KUKA KRL program: MyProgram_215().src

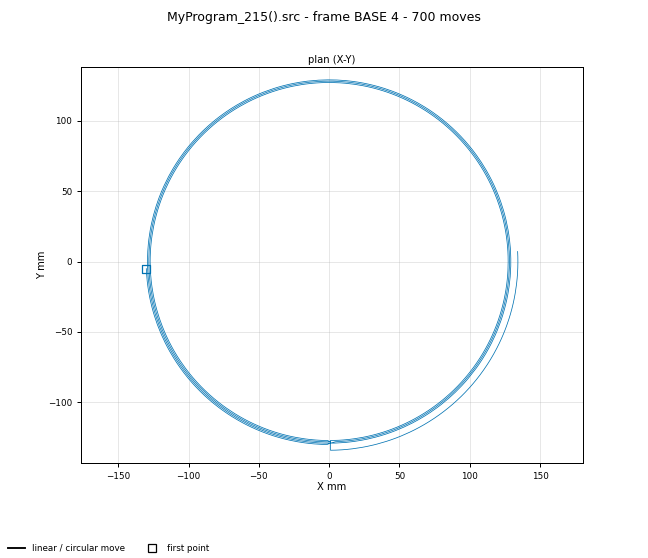
[picture p0: tool path of MyProgram_215().src in frame BASE 4, 700 of 700 moves have a stored position in this frame; points joined in program order, loops and branches not executed]
&ACCESS RVP
&REL 1
&PARAM TEMPLATE = C:\KRC\Roboter\Template\vorgabe
&PARAM EDITMASK = *
DEF MyProgram_215()
; ---- Setting reference (Base) ----
$BASE = BASE_DATA[4]

; --------------------------
; ---- Setting tool (TCP) ----
$TOOL = TOOL_DATA[3]
; --------------------------

$VEL.CP = VEL_APROX_PRINT
Startdeposition()
$VEL.CP = VEL_PRINT
LIN {X -130.0053,Y -5.0673,Z 151,A 179.9442,B 21.842,C -0.957,E1 21.7019,E2 267.4478} C_DIS
LIN {X -129.8507,Y -8.1164,Z 151,A -178.6124,B 21.842,C -0.9568,E1 21.7021,E2 265.9949} C_DIS
LIN {X -129.3313,Y -14.1597,Z 151,A -175.7971,B 21.8421,C -0.9542,E1 21.7029,E2 263.1669} C_DIS
LIN {X -128.8649,Y -17.9196,Z 151,A -174.1689,B 21.8424,C -0.9473,E1 21.7035,E2 261.5461} C_DIS
LIN {X -128.3149,Y -21.5014,Z 151,A -172.6656,B 21.8428,C -0.9385,E1 21.7041,E2 260.0561} C_DIS
LIN {X -127.7529,Y -24.622,Z 151,A -171.2515,B 21.8429,C -0.9349,E1 21.7049,E2 258.6421} C_DIS
LIN {X -127.1006,Y -27.7949,Z 151,A -169.6773,B 21.8429,C -0.9366,E1 21.7058,E2 257.0526} C_DIS
LIN {X -126.1184,Y -31.9552,Z 151,A -167.8984,B 21.8433,C -0.9266,E1 21.707,E2 255.2887} C_DIS
LIN {X -125.2346,Y -35.2609,Z 151,A -166.3979,B 21.8435,C -0.9217,E1 21.7081,E2 253.7911} C_DIS
LIN {X -124.2723,Y -38.5171,Z 151,A -164.8134,B 21.8435,C -0.9209,E1 21.7094,E2 252.1982} C_DIS
LIN {X -122.0887,Y -44.9645,Z 151,A -161.9059,B 21.844,C -0.9083,E1 21.712,E2 249.3057} C_DIS
LIN {X -120.3033,Y -49.5427,Z 151,A -159.7544,B 21.8443,C -0.9015,E1 21.7142,E2 247.1586} C_DIS
LIN {X -119.3188,Y -51.8654,Z 151,A -158.5882,B 21.8443,C -0.9006,E1 21.7155,E2 245.9873} C_DIS
LIN {X -117.9739,Y -54.8558,Z 151,A -157.1185,B 21.8444,C -0.8976,E1 21.7172,E2 244.5164} C_DIS
LIN {X -116.6239,Y -57.6698,Z 151,A -155.732,B 21.8446,C -0.8942,E1 21.7189,E2 243.1302} C_DIS
LIN {X -115.0398,Y -60.7689,Z 151,A -153.8793,B 21.8442,C -0.9033,E1 21.7214,E2 241.2414} C_DIS
LIN {X -113.4726,Y -63.6497,Z 151,A -152.4287,B 21.8443,C -0.8997,E1 21.7233,E2 239.7918} C_DIS
LIN {X -111.8624,Y -66.4401,Z 151,A -151.4946,B 21.8453,C -0.8757,E1 21.7246,E2 238.9168} C_DIS
LIN {X -110.3326,Y -68.9508,Z 151,A -149.9036,B 21.8449,C -0.8847,E1 21.727,E2 237.2922} C_DIS
LIN {X -108.359,Y -72.0127,Z 151,A -148.2536,B 21.845,C -0.8825,E1 21.7295,E2 235.6385} C_DIS
LIN {X -105.7262,Y -75.825,Z 151,A -146.2343,B 21.8452,C -0.8765,E1 21.7327,E2 233.6238} C_DIS
LIN {X -103.0748,Y -79.3925,Z 151,A -144.2157,B 21.8453,C -0.8743,E1 21.7361,E2 231.6} C_DIS
LIN {X -100.2325,Y -82.9511,Z 151,A -142.2432,B 21.8456,C -0.8682,E1 21.7396,E2 229.6333} C_DIS
LIN {X -97.3714,Y -86.2918,Z 151,A -140.1894,B 21.8456,C -0.8687,E1 21.7434,E2 227.5674} C_DIS
LIN {X -94.8101,Y -89.0985,Z 151,A -138.5955,B 21.8458,C -0.8616,E1 21.7464,E2 225.9844} C_DIS
LIN {X -91.7544,Y -92.2419,Z 151,A -136.1731,B 21.8452,C -0.8785,E1 21.7513,E2 223.5046} C_DIS
LIN {X -88.3402,Y -95.5175,Z 151,A -134.5958,B 21.8461,C -0.8526,E1 21.7544,E2 221.9896} C_DIS
LIN {X -85.1915,Y -98.3361,Z 151,A -132.7072,B 21.8462,C -0.8501,E1 21.7584,E2 220.0991} C_DIS
LIN {X -81.9083,Y -101.0868,Z 151,A -130.7823,B 21.8463,C -0.8482,E1 21.7625,E2 218.1708} C_DIS
LIN {X -78.3266,Y -103.8864,Z 151,A -128.5806,B 21.8461,C -0.8532,E1 21.7675,E2 215.9463} C_DIS
LIN {X -75.6688,Y -105.8379,Z 151,A -127.3113,B 21.8465,C -0.8429,E1 21.7703,E2 214.6997} C_DIS
LIN {X -72.1973,Y -108.2357,Z 151,A -125.4781,B 21.8466,C -0.8388,E1 21.7745,E2 212.8705} C_DIS
LIN {X -69.0452,Y -110.2738,Z 151,A -123.8621,B 21.8468,C -0.8347,E1 21.7783,E2 211.2596} C_DIS
LIN {X -65.5088,Y -112.4107,Z 151,A -121.9616,B 21.8468,C -0.8355,E1 21.7829,E2 209.3502} C_DIS
LIN {X -61.4607,Y -114.6736,Z 151,A -119.7151,B 21.8465,C -0.8416,E1 21.7885,E2 207.0798} C_DIS
LIN {X -58.5733,Y -116.1738,Z 151,A -118.6176,B 21.8471,C -0.8253,E1 21.7911,E2 206.023} C_DIS
LIN {X -55.1563,Y -117.835,Z 151,A -116.7367,B 21.8469,C -0.8323,E1 21.7959,E2 204.1176} C_DIS
LIN {X -51.0969,Y -119.6511,Z 151,A -114.7006,B 21.8469,C -0.8335,E1 21.8011,E2 202.0725} C_DIS
LIN {X -46.9474,Y -121.3381,Z 151,A -112.9585,B 21.8473,C -0.8215,E1 21.8056,E2 200.3584} C_DIS
LIN {X -42.9787,Y -122.8004,Z 151,A -111.0488,B 21.8473,C -0.8219,E1 21.8106,E2 198.4432} C_DIS
LIN {X -39.5704,Y -123.9401,Z 151,A -109.5332,B 21.8474,C -0.8177,E1 21.8146,E2 196.9357} C_DIS
LIN {X -36.3158,Y -124.9328,Z 151,A -108.0119,B 21.8474,C -0.8177,E1 21.8187,E2 195.4116} C_DIS
LIN {X -32.514,Y -125.9766,Z 151,A -105.7713,B 21.8466,C -0.8389,E1 21.8249,E2 193.1101} C_DIS
LIN {X -28.2456,Y -127.0028,Z 151,A -104.3076,B 21.8474,C -0.8171,E1 21.8288,E2 191.7029} C_DIS
LIN {X -22.4235,Y -128.1579,Z 151,A -101.5355,B 21.8472,C -0.823,E1 21.8364,E2 188.9112} C_DIS
LIN {X -18.2657,Y -128.8154,Z 151,A -99.8848,B 21.8476,C -0.8135,E1 21.8409,E2 187.2845} C_DIS
LIN {X -14.3497,Y -129.3109,Z 151,A -97.7475,B 21.8469,C -0.8311,E1 21.847,E2 185.0985} C_DIS
LIN {X -10.6851,Y -129.6647,Z 151,A -96.279,B 21.8472,C -0.8241,E1 21.851,E2 183.6479} C_DIS
LIN {X -5.5701,Y -129.9857,Z 151,A -94.1837,B 21.8474,C -0.8169,E1 21.8568,E2 181.5713} C_DIS
LIN {X -1.5263,Y -130.0967,Z 151,A -92.0677,B 21.8469,C -0.8323,E1 21.8628,E2 179.414} C_DIS
LIN {X -1.5263,Y -130.0967,Z 151,A -92.0677,B 21.8469,C -0.8323,E1 21.8628,E2 179.414} C_DIS
Enddeposition()
LIN {X 0.9297,Y -129.1307,Z 151,A -91.5034,B 20.7332,C -0.6398,E1 20.7439,E2 179.2548} C_DIS
Startdeposition()
$VEL.CP = VEL_PRINT
LIN {X -3.6627,Y -129.1076,Z 151,A -93.7153,B 20.7334,C -0.6318,E1 20.7376,E2 181.4893} C_DIS
LIN {X -8.0279,Y -128.9098,Z 151,A -95.6805,B 20.7334,C -0.6306,E1 20.7322,E2 183.4585} C_DIS
LIN {X -14.7037,Y -128.3212,Z 151,A -98.7805,B 20.7336,C -0.6256,E1 20.7235,E2 186.5747} C_DIS
LIN {X -20.0176,Y -127.599,Z 151,A -100.965,B 20.7333,C -0.6342,E1 20.7175,E2 188.7369} C_DIS
LIN {X -23.6572,Y -126.9757,Z 151,A -102.7964,B 20.7335,C -0.6269,E1 20.7124,E2 190.5914} C_DIS
LIN {X -28.0811,Y -126.0716,Z 151,A -105.0426,B 20.7338,C -0.6179,E1 20.7062,E2 192.8664} C_DIS
LIN {X -31.2653,Y -125.3191,Z 151,A -106.2307,B 20.7335,C -0.6294,E1 20.7031,E2 194.0238} C_DIS
LIN {X -34.6603,Y -124.4218,Z 151,A -107.7187,B 20.7333,C -0.6333,E1 20.6991,E2 195.5037} C_DIS
LIN {X -37.6238,Y -123.558,Z 151,A -109.1075,B 20.7333,C -0.6335,E1 20.6953,E2 196.8949} C_DIS
LIN {X -40.9396,Y -122.4992,Z 151,A -110.671,B 20.7333,C -0.6339,E1 20.6912,E2 198.4607} C_DIS
LIN {X -44.9395,Y -121.0895,Z 151,A -112.5539,B 20.7333,C -0.6355,E1 20.6862,E2 200.3437} C_DIS
LIN {X -49.6607,Y -119.2304,Z 151,A -114.8055,B 20.7333,C -0.6377,E1 20.6804,E2 202.595} C_DIS
LIN {X -53.9707,Y -117.3426,Z 151,A -116.9258,B 20.7332,C -0.6387,E1 20.675,E2 204.7188} C_DIS
LIN {X -56.9619,Y -115.9199,Z 151,A -118.3817,B 20.7332,C -0.641,E1 20.6713,E2 206.1728} C_DIS
LIN {X -62.2333,Y -113.18,Z 151,A -121.1366,B 20.7332,C -0.6397,E1 20.6645,E2 208.941} C_DIS
LIN {X -66.0389,Y -111.0019,Z 151,A -122.937,B 20.7329,C -0.6482,E1 20.6602,E2 210.7237} C_DIS
LIN {X -69.6038,Y -108.802,Z 151,A -124.8823,B 20.7329,C -0.6476,E1 20.6556,E2 212.6785} C_DIS
LIN {X -73.1285,Y -106.4649,Z 151,A -126.7619,B 20.7329,C -0.6505,E1 20.6512,E2 214.5576} C_DIS
LIN {X -77.9911,Y -102.9563,Z 151,A -129.4785,B 20.7328,C -0.6528,E1 20.6451,E2 217.2795} C_DIS
LIN {X -81.4308,Y -100.2583,Z 151,A -131.4493,B 20.7328,C -0.6551,E1 20.6408,E2 219.2528} C_DIS
LIN {X -84.7969,Y -97.4272,Z 151,A -133.3793,B 20.7326,C -0.6596,E1 20.6367,E2 221.1791} C_DIS
LIN {X -87.2832,Y -95.2062,Z 151,A -135.0805,B 20.7327,C -0.6539,E1 20.6331,E2 222.9049} C_DIS
LIN {X -89.6382,Y -92.9921,Z 151,A -136.651,B 20.7328,C -0.6515,E1 20.63,E2 224.4901} C_DIS
LIN {X -92.4164,Y -90.2322,Z 151,A -137.976,B 20.7322,C -0.6712,E1 20.6275,E2 225.7662} C_DIS
LIN {X -94.6886,Y -87.8446,Z 151,A -139.5529,B 20.7322,C -0.6699,E1 20.6244,E2 227.3553} C_DIS
LIN {X -97.6329,Y -84.5606,Z 151,A -141.5197,B 20.7322,C -0.6739,E1 20.6208,E2 229.3216} C_DIS
LIN {X -100.4671,Y -81.1722,Z 151,A -143.4289,B 20.7319,C -0.6804,E1 20.6174,E2 231.2232} C_DIS
LIN {X -103.0369,Y -77.8843,Z 151,A -145.3108,B 20.7319,C -0.6837,E1 20.6142,E2 233.107} C_DIS
LIN {X -105.6551,Y -74.2939,Z 151,A -147.2947,B 20.7317,C -0.688,E1 20.611,E2 235.0904} C_DIS
LIN {X -108.1691,Y -70.5839,Z 151,A -149.3281,B 20.7316,C -0.6913,E1 20.6078,E2 237.127} C_DIS
LIN {X -110.4376,Y -66.9785,Z 151,A -151.1709,B 20.7314,C -0.698,E1 20.6051,E2 238.9624} C_DIS
LIN {X -111.9833,Y -64.3618,Z 151,A -153.0329,B 20.7319,C -0.682,E1 20.6025,E2 240.882} C_DIS
LIN {X -114.1086,Y -60.5108,Z 151,A -154.5183,B 20.7311,C -0.705,E1 20.6006,E2 242.3117} C_DIS
LIN {X -115.7032,Y -57.4013,Z 151,A -156.017,B 20.7309,C -0.7112,E1 20.5987,E2 243.8026} C_DIS
LIN {X -117.1677,Y -54.349,Z 151,A -157.5382,B 20.7309,C -0.7146,E1 20.5969,E2 245.3242} C_DIS
LIN {X -118.5542,Y -51.254,Z 151,A -158.9864,B 20.7306,C -0.721,E1 20.5953,E2 246.7641} C_DIS
LIN {X -120.7634,Y -45.8103,Z 151,A -161.7172,B 20.7306,C -0.7237,E1 20.5924,E2 249.506} C_DIS
LIN {X -122.8848,Y -39.77,Z 151,A -164.5633,B 20.7302,C -0.7318,E1 20.5899,E2 252.3491} C_DIS
LIN {X -123.9274,Y -36.3883,Z 151,A -166.0964,B 20.73,C -0.7379,E1 20.5886,E2 253.8758} C_DIS
LIN {X -124.8503,Y -33.0839,Z 151,A -167.6613,B 20.73,C -0.7408,E1 20.5875,E2 255.4435} C_DIS
LIN {X -125.8593,Y -29.0106,Z 151,A -169.5242,B 20.7298,C -0.7464,E1 20.5863,E2 257.304} C_DIS
LIN {X -126.609,Y -25.5407,Z 151,A -171.1471,B 20.7296,C -0.7494,E1 20.5853,E2 258.9302} C_DIS
LIN {X -127.3745,Y -21.3985,Z 151,A -172.9926,B 20.7294,C -0.756,E1 20.5844,E2 260.7703} C_DIS
LIN {X -127.9861,Y -17.38,Z 151,A -175.5299,B 20.7302,C -0.7341,E1 20.5835,E2 263.3887} C_DIS
LIN {X -128.5912,Y -12.1049,Z 151,A -177.2563,B 20.7291,C -0.765,E1 20.583,E2 265.04} C_DIS
LIN {X -128.8936,Y -8.2915,Z 151,A -178.9563,B 20.7289,C -0.7702,E1 20.5826,E2 266.7377} C_DIS
LIN {X -129.0916,Y -4.2397,Z 151,A 179.2339,B 20.7287,C -0.7754,E1 20.5824,E2 268.546} C_DIS
LIN {X -129.1578,Y 0.8597,Z 151,A 176.6799,B 20.7289,C -0.7717,E1 20.5824,E2 271.1298} C_DIS
LIN {X -129.0884,Y 4.3415,Z 151,A 175.416,B 20.7283,C -0.7871,E1 20.5825,E2 272.3593} C_DIS
LIN {X -128.9527,Y 7.3319,Z 151,A 173.8225,B 20.7285,C -0.7813,E1 20.5828,E2 273.9809} C_DIS
LIN {X -128.5432,Y 12.6046,Z 151,A 171.4465,B 20.7283,C -0.7876,E1 20.5834,E2 276.3565} C_DIS
LIN {X -128.17,Y 15.9693,Z 151,A 170.1984,B 20.7278,C -0.8018,E1 20.5838,E2 277.5734} C_DIS
LIN {X -127.6557,Y 19.6512,Z 151,A 168.5632,B 20.7276,C -0.8076,E1 20.5844,E2 279.2042} C_DIS
LIN {X -127.2111,Y 22.3523,Z 151,A 166.8372,B 20.7281,C -0.7923,E1 20.5853,E2 280.9865} C_DIS
LIN {X -126.3821,Y 26.6474,Z 151,A 165.3428,B 20.7273,C -0.815,E1 20.5861,E2 282.4272} C_DIS
LIN {X -125.5883,Y 30.1612,Z 151,A 163.8397,B 20.727,C -0.8235,E1 20.587,E2 283.9167} C_DIS
LIN {X -124.8371,Y 33.1334,Z 151,A 162.449,B 20.7268,C -0.8266,E1 20.588,E2 285.3088} C_DIS
LIN {X -123.0875,Y 39.1355,Z 151,A 159.643,B 20.7266,C -0.8339,E1 20.5903,E2 288.114} C_DIS
LIN {X -122.0484,Y 42.2644,Z 151,A 158.3319,B 20.7262,C -0.844,E1 20.5914,E2 289.4054} C_DIS
LIN {X -121.1749,Y 44.7115,Z 151,A 156.9214,B 20.7264,C -0.8378,E1 20.5928,E2 290.8435} C_DIS
LIN {X -119.8659,Y 48.1068,Z 151,A 155.3824,B 20.7261,C -0.8455,E1 20.5943,E2 292.3713} C_DIS
LIN {X -118.6442,Y 51.0458,Z 151,A 154.0106,B 20.7259,C -0.8512,E1 20.5958,E2 293.7361} C_DIS
LIN {X -117.3376,Y 53.9816,Z 151,A 152.3415,B 20.7261,C -0.8462,E1 20.5978,E2 295.4307} C_DIS
LIN {X -114.0661,Y 60.5917,Z 151,A 149.1729,B 20.7256,C -0.8595,E1 20.6018,E2 298.5823} C_DIS
LIN {X -110.7434,Y 66.4726,Z 151,A 146.0823,B 20.7254,C -0.8644,E1 20.6061,E2 301.6789} C_DIS
LIN {X -108.892,Y 69.4632,Z 151,A 144.3697,B 20.7254,C -0.8629,E1 20.6086,E2 303.4064} C_DIS
LIN {X -106.2606,Y 73.4261,Z 151,A 142.3324,B 20.7251,C -0.8714,E1 20.6118,E2 305.4322} C_DIS
LIN {X -103.1907,Y 77.6804,Z 151,A 140.0564,B 20.7248,C -0.8795,E1 20.6156,E2 307.6988} C_DIS
LIN {X -100.4877,Y 81.1467,Z 151,A 138.1128,B 20.7245,C -0.8847,E1 20.6189,E2 309.6386} C_DIS
LIN {X -97.6713,Y 84.516,Z 151,A 136.1657,B 20.7243,C -0.8897,E1 20.6224,E2 311.5827} C_DIS
LIN {X -92.7127,Y 89.9274,Z 151,A 132.8628,B 20.7241,C -0.8957,E1 20.6287,E2 314.8862} C_DIS
LIN {X -89.5873,Y 93.0418,Z 151,A 130.9978,B 20.7238,C -0.9038,E1 20.6324,E2 316.7379} C_DIS
LIN {X -86.0666,Y 96.3074,Z 151,A 128.5072,B 20.7241,C -0.8948,E1 20.6376,E2 319.2664} C_DIS
LIN {X -83.5065,Y 98.5355,Z 151,A 127.2562,B 20.7236,C -0.9078,E1 20.6402,E2 320.4865} C_DIS
LIN {X -80.5766,Y 100.9455,Z 151,A 125.2849,B 20.7239,C -0.9003,E1 20.6446,E2 322.4882} C_DIS
LIN {X -77.8539,Y 103.0595,Z 151,A 123.9356,B 20.7235,C -0.9103,E1 20.6475,E2 323.8151} C_DIS
LIN {X -73.6245,Y 106.1226,Z 151,A 121.6955,B 20.7232,C -0.9178,E1 20.6526,E2 326.0434} C_DIS
LIN {X -70.0292,Y 108.5293,Z 151,A 120.0278,B 20.7226,C -0.9311,E1 20.6564,E2 327.68} C_DIS
LIN {X -65.7465,Y 111.176,Z 151,A 117.5115,B 20.7229,C -0.9241,E1 20.6625,E2 330.2259} C_DIS
LIN {X -59.9533,Y 114.4013,Z 151,A 114.674,B 20.7225,C -0.933,E1 20.6694,E2 333.0481} C_DIS
LIN {X -56.9239,Y 115.9387,Z 151,A 113.1648,B 20.7225,C -0.9353,E1 20.6732,E2 334.5558} C_DIS
LIN {X -53.8667,Y 117.3907,Z 151,A 111.5145,B 20.7225,C -0.9316,E1 20.6774,E2 336.2214} C_DIS
LIN {X -50.1887,Y 119.0099,Z 151,A 109.7546,B 20.7225,C -0.935,E1 20.6819,E2 337.9769} C_DIS
LIN {X -46.6923,Y 120.4239,Z 151,A 108.1581,B 20.7222,C -0.9402,E1 20.686,E2 339.5629} C_DIS
LIN {X -39.5979,Y 122.9398,Z 151,A 104.8024,B 20.7221,C -0.9435,E1 20.6949,E2 342.9173} C_DIS
LIN {X -36.2796,Y 123.9592,Z 151,A 103.286,B 20.722,C -0.946,E1 20.6989,E2 344.4296} C_DIS
LIN {X -33.094,Y 124.8476,Z 151,A 101.7573,B 20.722,C -0.945,E1 20.703,E2 345.9641} C_DIS
LIN {X -28.8799,Y 125.8892,Z 151,A 99.9263,B 20.7218,C -0.9505,E1 20.708,E2 347.7826} C_DIS
LIN {X -26.0513,Y 126.5051,Z 151,A 97.8758,B 20.723,C -0.9211,E1 20.7138,E2 349.9193} C_DIS
LIN {X -20.9039,Y 127.457,Z 151,A 96.4813,B 20.7214,C -0.9596,E1 20.7174,E2 351.2065} C_DIS
LIN {X -15.5852,Y 128.216,Z 151,A 93.9463,B 20.7216,C -0.9549,E1 20.7244,E2 353.7573} C_DIS
LIN {X -7.6009,Y 128.9361,Z 151,A 89.3024,B 20.7234,C -0.9128,E1 20.7377,E2 358.5226} C_DIS
LIN {X -0.8821,Y 129.1567,Z 151,A 87.1493,B 20.7219,C -0.9466,E1 20.7434,E2 360.5802} C_DIS
LIN {X 5.5468,Y 129.0414,Z 151,A 84.3233,B 20.7219,C -0.9478,E1 20.7513,E2 363.402} C_DIS
LIN {X 11.5803,Y 128.6413,Z 151,A 81.092,B 20.7229,C -0.9253,E1 20.7605,E2 366.6948} C_DIS
LIN {X 16.6384,Y 128.0833,Z 151,A 79.5352,B 20.7216,C -0.9533,E1 20.7646,E2 368.1709} C_DIS
LIN {X 20.3991,Y 127.5399,Z 151,A 77.7174,B 20.7219,C -0.9473,E1 20.7696,E2 370.0035} C_DIS
LIN {X 24.1839,Y 126.875,Z 151,A 76.3281,B 20.7214,C -0.9597,E1 20.7733,E2 371.3561} C_DIS
LIN {X 28.1638,Y 126.0528,Z 151,A 74.243,B 20.7219,C -0.947,E1 20.7791,E2 373.4736} C_DIS
LIN {X 31.6138,Y 125.2306,Z 151,A 72.7307,B 20.7219,C -0.9486,E1 20.7832,E2 374.9786} C_DIS
LIN {X 35.4917,Y 124.1893,Z 151,A 70.8764,B 20.722,C -0.9443,E1 20.7882,E2 376.8413} C_DIS
LIN {X 39.2919,Y 123.0375,Z 151,A 69.2677,B 20.7218,C -0.9493,E1 20.7924,E2 378.4323} C_DIS
LIN {X 42.2556,Y 122.0514,Z 151,A 67.8648,B 20.7218,C -0.9474,E1 20.7962,E2 379.8373} C_DIS
LIN {X 44.7376,Y 121.1651,Z 151,A 66.6455,B 20.722,C -0.9442,E1 20.7994,E2 381.0625} C_DIS
LIN {X 48.8415,Y 119.5698,Z 151,A 64.5302,B 20.7224,C -0.9354,E1 20.8049,E2 383.1967} C_DIS
LIN {X 52.6173,Y 117.9555,Z 151,A 62.9351,B 20.7221,C -0.9429,E1 20.8089,E2 384.7659} C_DIS
LIN {X 55.5611,Y 116.5977,Z 151,A 61.0349,B 20.723,C -0.9217,E1 20.8139,E2 386.7197} C_DIS
LIN {X 59.2362,Y 114.7764,Z 151,A 59.5349,B 20.7225,C -0.9328,E1 20.8175,E2 388.1835} C_DIS
LIN {X 63.3196,Y 112.5753,Z 151,A 57.7241,B 20.7222,C -0.9404,E1 20.8219,E2 389.9663} C_DIS
LIN {X 67.7408,Y 109.9718,Z 151,A 55.2985,B 20.7226,C -0.9306,E1 20.8277,E2 392.4102} C_DIS
LIN {X 70.7847,Y 108.0377,Z 151,A 53.3664,B 20.7233,C -0.914,E1 20.8323,E2 394.3814} C_DIS
LIN {X 73.8306,Y 105.9793,Z 151,A 52.0652,B 20.7229,C -0.9253,E1 20.8352,E2 395.6453} C_DIS
LIN {X 77.4332,Y 103.3769,Z 151,A 50.0794,B 20.723,C -0.9212,E1 20.8397,E2 397.6338} C_DIS
LIN {X 80.8,Y 100.7673,Z 151,A 48.1634,B 20.7232,C -0.9166,E1 20.8439,E2 399.5539} C_DIS
LIN {X 84.2434,Y 97.9061,Z 151,A 46.2248,B 20.7232,C -0.9148,E1 20.848,E2 401.4883} C_DIS
LIN {X 87.6418,Y 94.8766,Z 151,A 44.2384,B 20.7234,C -0.9122,E1 20.8522,E2 403.4722} C_DIS
LIN {X 90.5991,Y 92.0565,Z 151,A 42.414,B 20.7236,C -0.9079,E1 20.8558,E2 405.2992} C_DIS
LIN {X 93.6216,Y 88.9813,Z 151,A 40.5101,B 20.7237,C -0.9042,E1 20.8595,E2 407.2037} C_DIS
LIN {X 96.4884,Y 85.8645,Z 151,A 38.6013,B 20.724,C -0.8987,E1 20.8631,E2 409.1176} C_DIS
LIN {X 99.3142,Y 82.5791,Z 151,A 36.7128,B 20.724,C -0.8957,E1 20.8665,E2 411.0038} C_DIS
LIN {X 102.1643,Y 79.0254,Z 151,A 34.7333,B 20.7242,C -0.8927,E1 20.8699,E2 412.9803} C_DIS
LIN {X 104.7829,Y 75.5196,Z 151,A 32.9678,B 20.7242,C -0.8956,E1 20.8728,E2 414.7272} C_DIS
LIN {X 108.2539,Y 70.4532,Z 151,A 30.126,B 20.7246,C -0.8835,E1 20.8773,E2 417.5855} C_DIS
LIN {X 111.5876,Y 65.0455,Z 151,A 27.2897,B 20.7249,C -0.8754,E1 20.8814,E2 420.4271} C_DIS
LIN {X 113.6663,Y 61.3399,Z 151,A 25.372,B 20.7252,C -0.8688,E1 20.884,E2 422.3507} C_DIS
LIN {X 115.2925,Y 58.2226,Z 151,A 23.6149,B 20.7257,C -0.8559,E1 20.8862,E2 424.1325} C_DIS
LIN {X 116.8357,Y 55.063,Z 151,A 22.3015,B 20.7254,C -0.8624,E1 20.8878,E2 425.4191} C_DIS
LIN {X 118.1209,Y 52.2474,Z 151,A 20.974,B 20.7255,C -0.8605,E1 20.8893,E2 426.743} C_DIS
LIN {X 120.5192,Y 46.4471,Z 151,A 18.1623,B 20.7259,C -0.8513,E1 20.8922,E2 429.5614} C_DIS
LIN {X 121.9865,Y 42.4427,Z 151,A 16.4267,B 20.7259,C -0.8527,E1 20.8939,E2 431.2811} C_DIS
LIN {X 123.0107,Y 39.376,Z 151,A 15.0997,B 20.7259,C -0.8532,E1 20.895,E2 432.5974} C_DIS
LIN {X 123.9103,Y 36.4468,Z 151,A 13.6468,B 20.7261,C -0.845,E1 20.8962,E2 434.0632} C_DIS
LIN {X 124.7602,Y 33.4218,Z 151,A 12.2598,B 20.7263,C -0.8411,E1 20.8972,E2 435.4513} C_DIS
LIN {X 125.7535,Y 29.4736,Z 151,A 10.4527,B 20.7265,C -0.8356,E1 20.8984,E2 437.2612} C_DIS
LIN {X 127.2146,Y 22.3331,Z 151,A 7.3801,B 20.7266,C -0.8328,E1 20.9001,E2 440.3196} C_DIS
LIN {X 127.6938,Y 19.4056,Z 151,A 5.4025,B 20.7279,C -0.7993,E1 20.901,E2 442.3766} C_DIS
LIN {X 128.282,Y 15.0319,Z 151,A 3.2696,B 20.7284,C -0.7855,E1 20.9017,E2 444.5328} C_DIS
LIN {X 128.7977,Y 9.6649,Z 151,A 1.5986,B 20.7275,C -0.8099,E1 20.902,E2 446.1232} C_DIS
LIN {X 128.9879,Y 6.6592,Z 151,A -0.3127,B 20.7286,C -0.7802,E1 20.9023,E2 448.1039} C_DIS
LIN {X 129.1467,Y 1.8462,Z 151,A -2.4888,B 20.7289,C -0.7717,E1 20.9023,E2 450.288} C_DIS
LIN {X 129.1192,Y -3.2456,Z 151,A -4.0845,B 20.7281,C -0.7939,E1 20.9023,E2 451.8096} C_DIS
LIN {X 128.6983,Y -10.9049,Z 151,A -7.09,B 20.7278,C -0.8009,E1 20.9018,E2 454.7736} C_DIS
LIN {X 127.9573,Y -17.5936,Z 151,A -10.4752,B 20.7288,C -0.7734,E1 20.9008,E2 458.2112} C_DIS
LIN {X 127.1175,Y -22.8758,Z 151,A -12.8779,B 20.7291,C -0.7646,E1 20.8996,E2 460.6213} C_DIS
LIN {X 126.3307,Y -26.8853,Z 151,A -14.5725,B 20.7291,C -0.7642,E1 20.8987,E2 462.3049} C_DIS
LIN {X 125.6489,Y -29.91,Z 151,A -15.9439,B 20.7293,C -0.7601,E1 20.8978,E2 463.6781} C_DIS
LIN {X 124.575,Y -34.1124,Z 151,A -18.3948,B 20.7303,C -0.7307,E1 20.896,E2 466.1942} C_DIS
LIN {X 123.2794,Y -38.5342,Z 151,A -19.9953,B 20.7298,C -0.744,E1 20.8947,E2 467.7459} C_DIS
LIN {X 122.0822,Y -42.1669,Z 151,A -21.5221,B 20.7298,C -0.7465,E1 20.8934,E2 469.2553} C_DIS
LIN {X 119.5654,Y -48.8523,Z 151,A -24.7743,B 20.7302,C -0.7331,E1 20.8901,E2 472.5228} C_DIS
LIN {X 118.0279,Y -52.4554,Z 151,A -26.2213,B 20.7299,C -0.7409,E1 20.8885,E2 473.9381} C_DIS
LIN {X 115.4692,Y -57.8755,Z 151,A -29.1528,B 20.7306,C -0.7209,E1 20.885,E2 476.9063} C_DIS
LIN {X 113.5727,Y -61.5138,Z 151,A -30.9895,B 20.7308,C -0.7149,E1 20.8825,E2 478.748} C_DIS
LIN {X 111.2948,Y -65.5442,Z 151,A -33.0946,B 20.7311,C -0.7068,E1 20.8796,E2 480.8625} C_DIS
LIN {X 108.9733,Y -69.3361,Z 151,A -35.0225,B 20.7311,C -0.7033,E1 20.8767,E2 482.7883} C_DIS
LIN {X 106.3001,Y -73.3687,Z 151,A -37.0807,B 20.7313,C -0.7013,E1 20.8735,E2 484.8395} C_DIS
LIN {X 104.5609,Y -75.8259,Z 151,A -38.569,B 20.7316,C -0.691,E1 20.8711,E2 486.3479} C_DIS
LIN {X 98.7726,Y -83.2262,Z 151,A -42.2866,B 20.7313,C -0.7001,E1 20.8647,E2 490.0186} C_DIS
LIN {X 96.9618,Y -85.3284,Z 151,A -44.1372,B 20.7323,C -0.6697,E1 20.8611,E2 491.9443} C_DIS
LIN {X 94.2143,Y -88.3536,Z 151,A -45.2917,B 20.7315,C -0.6942,E1 20.8591,E2 493.0238} C_DIS
LIN {X 89.6177,Y -93.0125,Z 151,A -48.4469,B 20.7321,C -0.6761,E1 20.8528,E2 496.2133} C_DIS
LIN {X 84.9797,Y -97.2677,Z 151,A -51.0407,B 20.732,C -0.6785,E1 20.8475,E2 498.7875} C_DIS
LIN {X 79.4845,Y -101.8082,Z 151,A -54.2486,B 20.7323,C -0.6696,E1 20.8405,E2 502.0053} C_DIS
LIN {X 76.6021,Y -103.9937,Z 151,A -56.0337,B 20.7326,C -0.6585,E1 20.8365,E2 503.814} C_DIS
LIN {X 71.7873,Y -107.3738,Z 151,A -58.5474,B 20.7326,C -0.6575,E1 20.8307,E2 506.3197} C_DIS
LIN {X 68.3618,Y -109.5866,Z 151,A -60.3785,B 20.7328,C -0.6532,E1 20.8264,E2 508.1557} C_DIS
LIN {X 63.5548,Y -112.4431,Z 151,A -62.9324,B 20.733,C -0.6457,E1 20.8202,E2 510.7213} C_DIS
LIN {X 59.1082,Y -114.8416,Z 151,A -65.0469,B 20.733,C -0.6474,E1 20.815,E2 512.8234} C_DIS
LIN {X 55.9527,Y -116.4106,Z 151,A -66.6966,B 20.7331,C -0.6413,E1 20.8108,E2 514.485} C_DIS
LIN {X 53.2005,Y -117.6946,Z 151,A -68.8209,B 20.7341,C -0.6061,E1 20.8052,E2 516.7018} C_DIS
LIN {X 47.2666,Y -120.2001,Z 151,A -70.7691,B 20.7331,C -0.6409,E1 20.8004,E2 518.5466} C_DIS
LIN {X 44.4573,Y -121.2687,Z 151,A -72.1229,B 20.7332,C -0.6383,E1 20.7968,E2 519.9043} C_DIS
LIN {X 40.2341,Y -122.7341,Z 151,A -74.1051,B 20.7332,C -0.636,E1 20.7916,E2 521.8883} C_DIS
LIN {X 36.5336,Y -123.8849,Z 151,A -75.7703,B 20.7332,C -0.6364,E1 20.7872,E2 523.5487} C_DIS
LIN {X 32.859,Y -124.9103,Z 151,A -77.5961,B 20.7335,C -0.629,E1 20.7822,E2 525.3917} C_DIS
LIN {X 27.3988,Y -126.2198,Z 151,A -79.9348,B 20.7334,C -0.6332,E1 20.7759,E2 527.7146} C_DIS
LIN {X 23.3178,Y -127.0384,Z 151,A -82.5736,B 20.7343,C -0.5984,E1 20.7684,E2 530.4477} C_DIS
LIN {X 17.5674,Y -127.9611,Z 151,A -85.2005,B 20.7344,C -0.595,E1 20.7611,E2 533.0815} C_DIS
LIN {X 11.5745,Y -128.6418,Z 151,A -87.1227,B 20.7336,C -0.625,E1 20.756,E2 534.9175} C_DIS
LIN {X 4.2522,Y -129.0913,Z 151,A -90.1916,B 20.7334,C -0.6316,E1 20.7475,E2 537.9665} C_DIS
LIN {X 0.9297,Y -129.1307,Z 151,A -91.4997,B 20.7332,C -0.6385,E1 20.7439,E2 539.2548} C_DIS
Enddeposition()
LIN {X 0.9297,Y -129.1307,Z 151,A -91.4997,B 20.7332,C -0.6385,E1 20.7439,E2 539.2548} C_DIS
Startdeposition()
$VEL.CP = VEL_PRINT
LIN {X 4.5456,Y -128.1352,Z 151,A -88.007,B 19.4412,C -0.5334,E1 19.4588,E2 535.9333} C_DIS
LIN {X 11.5645,Y -127.6942,Z 151,A -85.1224,B 19.4415,C -0.5245,E1 19.4667,E2 533.0779} C_DIS
LIN {X 17.2176,Y -127.0549,Z 151,A -83.1506,B 19.442,C -0.5031,E1 19.472,E2 531.1724} C_DIS
LIN {X 23.2745,Y -126.0866,Z 151,A -80.6065,B 19.4422,C -0.4971,E1 19.479,E2 528.6497} C_DIS
LIN {X 26.989,Y -125.3421,Z 151,A -78.9497,B 19.4422,C -0.4971,E1 19.4835,E2 526.9957} C_DIS
LIN {X 30.6098,Y -124.5086,Z 151,A -76.9994,B 19.4418,C -0.5103,E1 19.4889,E2 525.0097} C_DIS
LIN {X 33.8013,Y -123.6813,Z 151,A -75.7687,B 19.442,C -0.5019,E1 19.4921,E2 523.8065} C_DIS
LIN {X 37.4014,Y -122.6383,Z 151,A -74.1267,B 19.442,C -0.5024,E1 19.4965,E2 522.1668} C_DIS
LIN {X 41.2225,Y -121.4095,Z 151,A -71.9487,B 19.4416,C -0.5201,E1 19.5024,E2 519.9415} C_DIS
LIN {X 44.7178,Y -120.164,Z 151,A -70.6985,B 19.442,C -0.5056,E1 19.5055,E2 518.7381} C_DIS
LIN {X 47.6944,Y -119.0138,Z 151,A -68.3734,B 19.441,C -0.5443,E1 19.5119,E2 516.3044} C_DIS
LIN {X 53.5461,Y -116.4983,Z 151,A -66.4896,B 19.4419,C -0.5089,E1 19.5164,E2 514.5326} C_DIS
LIN {X 56.4309,Y -115.1287,Z 151,A -64.9876,B 19.4417,C -0.5142,E1 19.5202,E2 513.0201} C_DIS
LIN {X 59.7815,Y -113.4247,Z 151,A -63.3722,B 19.4417,C -0.5142,E1 19.5241,E2 511.4105} C_DIS
LIN {X 62.8324,Y -111.7656,Z 151,A -61.8302,B 19.4417,C -0.5164,E1 19.5279,E2 509.8679} C_DIS
LIN {X 66.626,Y -109.547,Z 151,A -59.7625,B 19.4415,C -0.5241,E1 19.5329,E2 507.7856} C_DIS
LIN {X 69.9329,Y -107.4656,Z 151,A -58.1554,B 19.4415,C -0.5216,E1 19.5367,E2 506.1928} C_DIS
LIN {X 73.0014,Y -105.4056,Z 151,A -56.6169,B 19.4415,C -0.5201,E1 19.5402,E2 504.6656} C_DIS
LIN {X 75.194,Y -103.8524,Z 151,A -54.9085,B 19.441,C -0.5435,E1 19.5442,E2 502.8954} C_DIS
LIN {X 78.1485,Y -101.6483,Z 151,A -53.546,B 19.4412,C -0.535,E1 19.5471,E2 501.5647} C_DIS
LIN {X 81.5589,Y -98.9327,Z 151,A -51.5496,B 19.441,C -0.5411,E1 19.5515,E2 499.56} C_DIS
LIN {X 84.5676,Y -96.3738,Z 151,A -49.211,B 19.4403,C -0.569,E1 19.5566,E2 497.1504} C_DIS
LIN {X 88.6141,Y -92.6661,Z 151,A -47.5277,B 19.441,C -0.5424,E1 19.5598,E2 495.5556} C_DIS
LIN {X 94.2085,Y -86.9726,Z 151,A -43.5588,B 19.4403,C -0.5676,E1 19.5676,E2 491.534} C_DIS
LIN {X 96.7818,Y -84.1,Z 151,A -42.1737,B 19.4406,C -0.5577,E1 19.57,E2 490.1867} C_DIS
LIN {X 99.529,Y -80.8306,Z 151,A -40.4657,B 19.4406,C -0.5542,E1 19.573,E2 488.4997} C_DIS
LIN {X 102.2354,Y -77.3784,Z 151,A -38.3429,B 19.4404,C -0.566,E1 19.5767,E2 486.3548} C_DIS
LIN {X 104.5778,Y -74.1827,Z 151,A -36.6237,B 19.4403,C -0.5685,E1 19.5795,E2 484.6391} C_DIS
LIN {X 106.6575,Y -71.1592,Z 151,A -35.0178,B 19.4403,C -0.5715,E1 19.582,E2 483.0347} C_DIS
LIN {X 109.1036,Y -67.3498,Z 151,A -33.2023,B 19.4403,C -0.5684,E1 19.5847,E2 481.2407} C_DIS
LIN {X 111.868,Y -62.6502,Z 151,A -30.5433,B 19.4398,C -0.5845,E1 19.5885,E2 478.5518} C_DIS
LIN {X 114.003,Y -58.6737,Z 151,A -28.7275,B 19.4399,C -0.5818,E1 19.5908,E2 476.7566} C_DIS
LIN {X 115.8608,Y -54.9126,Z 151,A -26.7416,B 19.4396,C -0.5919,E1 19.5933,E2 474.7547} C_DIS
LIN {X 117.5726,Y -51.1443,Z 151,A -24.9649,B 19.4396,C -0.5942,E1 19.5953,E2 472.9837} C_DIS
LIN {X 118.7672,Y -48.3062,Z 151,A -23.5031,B 19.4393,C -0.6019,E1 19.5968,E2 471.5096} C_DIS
LIN {X 119.9696,Y -45.2367,Z 151,A -21.8827,B 19.439,C -0.6125,E1 19.5985,E2 469.8694} C_DIS
LIN {X 121.584,Y -40.6985,Z 151,A -19.9406,B 19.439,C -0.6101,E1 19.6002,E2 467.9489} C_DIS
LIN {X 122.5596,Y -37.6586,Z 151,A -18.4589,B 19.4389,C -0.6168,E1 19.6015,E2 466.4585} C_DIS
LIN {X 123.6986,Y -33.7373,Z 151,A -16.5641,B 19.4386,C -0.6253,E1 19.6029,E2 464.5526} C_DIS
LIN {X 124.7379,Y -29.6586,Z 151,A -14.8736,B 19.4386,C -0.6231,E1 19.604,E2 462.8816} C_DIS
LIN {X 125.5328,Y -26.0929,Z 151,A -13.1952,B 19.4385,C -0.63,E1 19.605,E2 461.1953} C_DIS
LIN {X 126.2058,Y -22.6087,Z 151,A -11.8421,B 19.4386,C -0.6252,E1 19.6057,E2 459.8672} C_DIS
LIN {X 126.8742,Y -18.4966,Z 151,A -9.8404,B 19.4383,C -0.6368,E1 19.6066,E2 457.8462} C_DIS
LIN {X 127.2781,Y -15.4735,Z 151,A -7.8975,B 19.4373,C -0.6657,E1 19.6072,E2 455.8324} C_DIS
LIN {X 127.7522,Y -10.8845,Z 151,A -6.6351,B 19.4382,C -0.6383,E1 19.6076,E2 454.6615} C_DIS
LIN {X 128.1516,Y -4.0644,Z 151,A -3.4296,B 19.4377,C -0.6542,E1 19.608,E2 451.4338} C_DIS
LIN {X 128.2153,Y 0.5713,Z 151,A -1.2836,B 19.4374,C -0.6638,E1 19.608,E2 449.276} C_DIS
LIN {X 128.0283,Y 6.9346,Z 151,A 1.6418,B 19.437,C -0.6761,E1 19.6077,E2 446.3369} C_DIS
LIN {X 127.3568,Y 14.8143,Z 151,A 5.0398,B 19.4368,C -0.6812,E1 19.6069,E2 442.95} C_DIS
LIN {X 126.5259,Y 20.7458,Z 151,A 7.6754,B 19.4366,C -0.6877,E1 19.6058,E2 440.3155} C_DIS
LIN {X 125.8098,Y 24.7261,Z 151,A 9.6617,B 19.4361,C -0.7007,E1 19.6047,E2 438.3057} C_DIS
LIN {X 124.8397,Y 29.233,Z 151,A 11.6311,B 19.4361,C -0.7031,E1 19.6035,E2 436.3443} C_DIS
LIN {X 123.9069,Y 32.9559,Z 151,A 13.076,B 19.4363,C -0.6969,E1 19.6025,E2 434.9288} C_DIS
LIN {X 123.0906,Y 35.8849,Z 151,A 14.4679,B 19.4361,C -0.7023,E1 19.6015,E2 433.5313} C_DIS
LIN {X 122.1645,Y 38.9209,Z 151,A 15.9144,B 19.4359,C -0.7077,E1 19.6002,E2 432.0797} C_DIS
LIN {X 121.1267,Y 42.0395,Z 151,A 17.3657,B 19.4358,C -0.7112,E1 19.5989,E2 430.6287} C_DIS
LIN {X 119.9404,Y 45.3146,Z 151,A 18.8583,B 19.4358,C -0.713,E1 19.5975,E2 429.1416} C_DIS
LIN {X 118.8365,Y 48.1344,Z 151,A 20.6444,B 19.4349,C -0.735,E1 19.5956,E2 427.303} C_DIS
LIN {X 117.39,Y 51.5667,Z 151,A 21.9032,B 19.4354,C -0.7226,E1 19.5942,E2 426.0901} C_DIS
LIN {X 115.7989,Y 55.0421,Z 151,A 23.5814,B 19.4352,C -0.7262,E1 19.5923,E2 424.4134} C_DIS
LIN {X 113.8269,Y 59.0155,Z 151,A 25.6489,B 19.4349,C -0.7351,E1 19.5896,E2 422.3338} C_DIS
LIN {X 112.0078,Y 62.4006,Z 151,A 27.3706,B 19.4347,C -0.7398,E1 19.5873,E2 420.6098} C_DIS
LIN {X 110.3139,Y 65.3484,Z 151,A 29.0603,B 19.4343,C -0.7509,E1 19.5849,E2 418.8986} C_DIS
LIN {X 107.7579,Y 69.4828,Z 151,A 31.0565,B 19.4344,C -0.7491,E1 19.5819,E2 416.9208} C_DIS
LIN {X 106.2291,Y 71.7973,Z 151,A 32.5911,B 19.4338,C -0.7645,E1 19.5795,E2 415.3505} C_DIS
LIN {X 104.0729,Y 74.8895,Z 151,A 33.9869,B 19.4341,C -0.7566,E1 19.5773,E2 413.9871} C_DIS
LIN {X 101.4371,Y 78.4219,Z 151,A 35.9047,B 19.4341,C -0.7592,E1 19.574,E2 412.0736} C_DIS
LIN {X 98.6685,Y 81.878,Z 151,A 37.8261,B 19.4339,C -0.7615,E1 19.5707,E2 410.1572} C_DIS
LIN {X 95.8725,Y 85.1352,Z 151,A 39.7799,B 19.4337,C -0.7672,E1 19.5671,E2 408.1978} C_DIS
LIN {X 92.9806,Y 88.2849,Z 151,A 41.7133,B 19.4335,C -0.7723,E1 19.5634,E2 406.2603} C_DIS
LIN {X 89.9484,Y 91.3718,Z 151,A 43.6203,B 19.4335,C -0.7753,E1 19.5596,E2 404.355} C_DIS
LIN {X 86.6462,Y 94.5088,Z 151,A 45.6265,B 19.4333,C -0.7782,E1 19.5555,E2 402.351} C_DIS
LIN {X 83.3365,Y 97.4404,Z 151,A 47.6303,B 19.4331,C -0.7832,E1 19.5513,E2 400.3427} C_DIS
LIN {X 79.8969,Y 100.2793,Z 151,A 49.5806,B 19.4331,C -0.7852,E1 19.5471,E2 398.3962} C_DIS
LIN {X 76.2687,Y 103.0664,Z 151,A 51.631,B 19.4329,C -0.789,E1 19.5425,E2 396.3442} C_DIS
LIN {X 73.1626,Y 105.2934,Z 151,A 53.3355,B 19.4328,C -0.7917,E1 19.5386,E2 394.6393} C_DIS
LIN {X 69.4916,Y 107.7522,Z 151,A 55.2355,B 19.4328,C -0.7919,E1 19.5342,E2 392.7471} C_DIS
LIN {X 66.2173,Y 109.7941,Z 151,A 56.9256,B 19.4328,C -0.7931,E1 19.5302,E2 391.0604} C_DIS
LIN {X 62.3476,Y 112.0371,Z 151,A 58.9847,B 19.4325,C -0.7984,E1 19.5251,E2 388.9937} C_DIS
LIN {X 58.4591,Y 114.1122,Z 151,A 60.6502,B 19.4329,C -0.7889,E1 19.5211,E2 387.3628} C_DIS
LIN {X 55.9492,Y 115.3656,Z 151,A 62.264,B 19.4323,C -0.8047,E1 19.517,E2 385.7071} C_DIS
LIN {X 52.2154,Y 117.1006,Z 151,A 63.8411,B 19.4326,C -0.7965,E1 19.513,E2 384.16} C_DIS
LIN {X 49.4708,Y 118.2862,Z 151,A 65.4156,B 19.4322,C -0.8074,E1 19.5089,E2 382.5579} C_DIS
LIN {X 46.1615,Y 119.6169,Z 151,A 67.1239,B 19.4319,C -0.8135,E1 19.5044,E2 380.8362} C_DIS
LIN {X 41.7597,Y 121.2237,Z 151,A 68.9661,B 19.4322,C -0.8055,E1 19.4997,E2 379.0231} C_DIS
LIN {X 37.8326,Y 122.5063,Z 151,A 70.8614,B 19.4321,C -0.8089,E1 19.4946,E2 377.1221} C_DIS
LIN {X 34.4724,Y 123.4936,Z 151,A 72.3785,B 19.4321,C -0.8081,E1 19.4905,E2 375.6107} C_DIS
LIN {X 30.3847,Y 124.5629,Z 151,A 74.2683,B 19.4321,C -0.8094,E1 19.4854,E2 373.721} C_DIS
LIN {X 27.1259,Y 125.3125,Z 151,A 75.7754,B 19.4321,C -0.8107,E1 19.4813,E2 372.2125} C_DIS
LIN {X 22.9917,Y 126.1372,Z 151,A 77.6125,B 19.4321,C -0.8097,E1 19.4763,E2 370.3813} C_DIS
LIN {X 19.8087,Y 126.6756,Z 151,A 79.0493,B 19.4321,C -0.81,E1 19.4723,E2 368.9454} C_DIS
LIN {X 16.2032,Y 127.1878,Z 151,A 80.6525,B 19.4321,C -0.8095,E1 19.4679,E2 367.3455} C_DIS
LIN {X 11.7551,Y 127.6759,Z 151,A 82.7746,B 19.4319,C -0.8146,E1 19.462,E2 365.21} C_DIS
LIN {X 7.7513,Y 127.9806,Z 151,A 84.4828,B 19.4319,C -0.8114,E1 19.4572,E2 363.5124} C_DIS
LIN {X 2.89,Y 128.1837,Z 151,A 86.9964,B 19.4315,C -0.8243,E1 19.4501,E2 360.9608} C_DIS
LIN {X -0.4585,Y 128.2145,Z 151,A 88.1904,B 19.432,C -0.8125,E1 19.4469,E2 359.8023} C_DIS
LIN {X -4.2543,Y 128.1462,Z 151,A 90.2602,B 19.4314,C -0.8264,E1 19.441,E2 357.6905} C_DIS
LIN {X -7.8876,Y 127.9722,Z 151,A 91.515,B 19.432,C -0.8118,E1 19.4376,E2 356.4792} C_DIS
LIN {X -13.7844,Y 127.4718,Z 151,A 94.1768,B 19.432,C -0.8113,E1 19.4302,E2 353.8171} C_DIS
LIN {X -18.011,Y 126.9436,Z 151,A 96.0549,B 19.432,C -0.8093,E1 19.425,E2 351.9433} C_DIS
LIN {X -23.146,Y 126.1096,Z 151,A 98.6467,B 19.4317,C -0.8178,E1 19.4178,E2 349.3225} C_DIS
LIN {X -26.308,Y 125.489,Z 151,A 99.927,B 19.432,C -0.8106,E1 19.4144,E2 348.0617} C_DIS
LIN {X -30.1023,Y 124.631,Z 151,A 101.5611,B 19.4322,C -0.8053,E1 19.41,E2 346.4409} C_DIS
LIN {X -34.0108,Y 123.6227,Z 151,A 103.435,B 19.4322,C -0.8062,E1 19.4049,E2 344.5606} C_DIS
LIN {X -37.2511,Y 122.6843,Z 151,A 104.8218,B 19.4324,C -0.8001,E1 19.4012,E2 343.1889} C_DIS
LIN {X -39.815,Y 121.8782,Z 151,A 106.3559,B 19.432,C -0.8112,E1 19.3971,E2 341.6178} C_DIS
LIN {X -44.4885,Y 120.2499,Z 151,A 108.3007,B 19.4325,C -0.7987,E1 19.392,E2 339.7057} C_DIS
LIN {X -47.8858,Y 118.9367,Z 151,A 109.835,B 19.4327,C -0.7932,E1 19.3881,E2 338.1836} C_DIS
LIN {X -50.7102,Y 117.7603,Z 151,A 111.2867,B 19.4327,C -0.7944,E1 19.3843,E2 336.7237} C_DIS
LIN {X -54.5305,Y 116.043,Z 151,A 113.4023,B 19.4324,C -0.8007,E1 19.3789,E2 334.5822} C_DIS
LIN {X -58.6572,Y 114.0114,Z 151,A 115.1834,B 19.4329,C -0.7875,E1 19.3745,E2 332.8348} C_DIS
LIN {X -62.0719,Y 112.1898,Z 151,A 116.9982,B 19.4329,C -0.7878,E1 19.37,E2 331.0122} C_DIS
LIN {X -65.5974,Y 110.1655,Z 151,A 118.8458,B 19.433,C -0.7858,E1 19.3656,E2 329.1632} C_DIS
LIN {X -69.6241,Y 107.6661,Z 151,A 120.9558,B 19.4332,C -0.7818,E1 19.3606,E2 327.0566} C_DIS
LIN {X -72.6609,Y 105.6403,Z 151,A 122.6234,B 19.4332,C -0.78,E1 19.3568,E2 325.3869} C_DIS
LIN {X -76.0181,Y 103.2508,Z 151,A 125.1121,B 19.4324,C -0.8001,E1 19.351,E2 322.8261} C_DIS
LIN {X -80.1295,Y 100.0942,Z 151,A 126.8443,B 19.4335,C -0.774,E1 19.3474,E2 321.1641} C_DIS
LIN {X -83.4266,Y 97.3631,Z 151,A 128.6102,B 19.4338,C -0.7646,E1 19.3436,E2 319.4176} C_DIS
LIN {X -85.6118,Y 95.4467,Z 151,A 130.0691,B 19.4338,C -0.7676,E1 19.3405,E2 317.9422} C_DIS
LIN {X -88.7428,Y 92.5431,Z 151,A 131.967,B 19.4338,C -0.7629,E1 19.3367,E2 316.0481} C_DIS
LIN {X -91.6937,Y 89.6201,Z 151,A 133.8256,B 19.434,C -0.7587,E1 19.333,E2 314.1917} C_DIS
LIN {X -95.267,Y 85.8125,Z 151,A 136.2167,B 19.4342,C -0.7552,E1 19.3285,E2 311.7974} C_DIS
LIN {X -98.106,Y 82.5513,Z 151,A 138.1648,B 19.4343,C -0.751,E1 19.325,E2 309.8502} C_DIS
LIN {X -100.9536,Y 79.0435,Z 151,A 140.2361,B 19.4345,C -0.7477,E1 19.3214,E2 307.7759} C_DIS
LIN {X -103.4473,Y 75.7506,Z 151,A 142.4688,B 19.4341,C -0.7568,E1 19.3176,E2 305.5015} C_DIS
LIN {X -105.9313,Y 72.2369,Z 151,A 143.8873,B 19.435,C -0.7336,E1 19.3155,E2 304.1438} C_DIS
LIN {X -107.9147,Y 69.2379,Z 151,A 145.5372,B 19.435,C -0.7309,E1 19.3129,E2 302.4914} C_DIS
LIN {X -110.1684,Y 65.5925,Z 151,A 147.8663,B 19.4347,C -0.7403,E1 19.3095,E2 300.1177} C_DIS
LIN {X -112.0891,Y 62.2537,Z 151,A 149.2307,B 19.4354,C -0.7228,E1 19.3077,E2 298.7969} C_DIS
LIN {X -113.9968,Y 58.6859,Z 151,A 151.2975,B 19.4352,C -0.7269,E1 19.305,E2 296.7032} C_DIS
LIN {X -115.438,Y 55.7976,Z 151,A 152.9735,B 19.4351,C -0.7311,E1 19.303,E2 295.0026} C_DIS
LIN {X -117.2472,Y 51.8877,Z 151,A 154.5135,B 19.4358,C -0.7118,E1 19.3013,E2 293.5098} C_DIS
LIN {X -118.8352,Y 48.1376,Z 151,A 156.2263,B 19.4361,C -0.7026,E1 19.2994,E2 291.8121} C_DIS
LIN {X -119.9954,Y 45.1678,Z 151,A 157.581,B 19.4363,C -0.6959,E1 19.2981,E2 290.4676} C_DIS
LIN {X -121.6783,Y 40.4153,Z 151,A 159.5432,B 19.4369,C -0.6789,E1 19.2963,E2 288.542} C_DIS
LIN {X -123.4977,Y 34.4578,Z 151,A 163.118,B 19.4362,C -0.6983,E1 19.2934,E2 284.8812} C_DIS
LIN {X -124.4543,Y 30.8331,Z 151,A 164.4794,B 19.4368,C -0.682,E1 19.2925,E2 283.5586} C_DIS
LIN {X -125.3319,Y 27.036,Z 151,A 166.132,B 19.4371,C -0.6736,E1 19.2915,E2 281.9189} C_DIS
LIN {X -126.1224,Y 23.0745,Z 151,A 168.0731,B 19.4371,C -0.6728,E1 19.2905,E2 279.965} C_DIS
LIN {X -126.7443,Y 19.3653,Z 151,A 169.6959,B 19.4373,C -0.6655,E1 19.2898,E2 278.3514} C_DIS
LIN {X -127.255,Y 15.6677,Z 151,A 171.2754,B 19.4376,C -0.6572,E1 19.2892,E2 276.7846} C_DIS
LIN {X -127.6197,Y 12.3407,Z 151,A 172.9079,B 19.4376,C -0.6573,E1 19.2887,E2 275.1387} C_DIS
LIN {X -127.9548,Y 8.1697,Z 151,A 174.7527,B 19.4378,C -0.6506,E1 19.2883,E2 273.2996} C_DIS
LIN {X -128.1276,Y 4.7423,Z 151,A 176.227,B 19.438,C -0.6437,E1 19.2882,E2 271.8343} C_DIS
LIN {X -128.1998,Y 1.9825,Z 151,A 177.5898,B 19.438,C -0.6444,E1 19.2881,E2 270.4586} C_DIS
LIN {X -128.1997,Y -1.994,Z 151,A 179.4394,B 19.4381,C -0.6415,E1 19.2881,E2 268.6033} C_DIS
LIN {X -128.0701,Y -6.1035,Z 151,A -178.775,B 19.4383,C -0.6339,E1 19.2883,E2 266.8263} C_DIS
LIN {X -127.8587,Y -9.5542,Z 151,A -177.2442,B 19.4385,C -0.6286,E1 19.2886,E2 265.2994} C_DIS
LIN {X -127.544,Y -13.1137,Z 151,A -175.7234,B 19.4387,C -0.621,E1 19.289,E2 263.7896} C_DIS
LIN {X -127.0374,Y -17.3504,Z 151,A -173.6706,B 19.4387,C -0.6203,E1 19.2897,E2 261.7228} C_DIS
LIN {X -126.4993,Y -20.9048,Z 151,A -172.0346,B 19.4389,C -0.6164,E1 19.2904,E2 260.0855} C_DIS
LIN {X -125.7729,Y -24.913,Z 151,A -170.1333,B 19.4389,C -0.6137,E1 19.2914,E2 258.1774} C_DIS
LIN {X -124.9917,Y -28.5677,Z 151,A -168.6129,B 19.4393,C -0.6034,E1 19.2923,E2 256.6765} C_DIS
LIN {X -124.2168,Y -31.769,Z 151,A -167.0151,B 19.4393,C -0.6035,E1 19.2934,E2 255.066} C_DIS
LIN {X -123.1346,Y -35.7347,Z 151,A -165.212,B 19.4395,C -0.5969,E1 19.2948,E2 253.2692} C_DIS
LIN {X -122.1414,Y -38.9933,Z 151,A -163.5264,B 19.4395,C -0.5982,E1 19.2962,E2 251.5667} C_DIS
LIN {X -120.7015,Y -43.246,Z 151,A -161.7109,B 19.4398,C -0.5856,E1 19.2979,E2 249.7758} C_DIS
LIN {X -119.6672,Y -46.032,Z 151,A -160.4928,B 19.44,C -0.5779,E1 19.299,E2 248.572} C_DIS
LIN {X -118.5692,Y -48.7931,Z 151,A -158.9339,B 19.4399,C -0.5824,E1 19.3007,E2 246.988} C_DIS
LIN {X -117.1319,Y -52.1454,Z 151,A -157.2807,B 19.4399,C -0.5787,E1 19.3026,E2 245.334} C_DIS
LIN {X -115.4286,Y -55.8173,Z 151,A -155.4051,B 19.4401,C -0.5761,E1 19.3048,E2 243.4527} C_DIS
LIN {X -113.776,Y -59.1125,Z 151,A -153.9877,B 19.4404,C -0.5634,E1 19.3066,E2 242.0637} C_DIS
LIN {X -111.8542,Y -62.6747,Z 151,A -152.0348,B 19.4404,C -0.5637,E1 19.3092,E2 240.096} C_DIS
LIN {X -110.1248,Y -65.6658,Z 151,A -150.4773,B 19.4405,C -0.5602,E1 19.3114,E2 238.5385} C_DIS
LIN {X -108.2361,Y -68.7353,Z 151,A -148.7418,B 19.4405,C -0.5606,E1 19.314,E2 236.7902} C_DIS
LIN {X -106.31,Y -71.6777,Z 151,A -147.1786,B 19.4406,C -0.5564,E1 19.3164,E2 235.2294} C_DIS
LIN {X -103.7023,Y -75.4011,Z 151,A -145.207,B 19.4408,C -0.5493,E1 19.3196,E2 233.2667} C_DIS
LIN {X -101.1312,Y -78.8166,Z 151,A -143.2322,B 19.4408,C -0.5471,E1 19.323,E2 231.2861} C_DIS
LIN {X -98.4881,Y -82.0958,Z 151,A -141.3054,B 19.441,C -0.5444,E1 19.3264,E2 229.3556} C_DIS
LIN {X -95.6803,Y -85.351,Z 151,A -139.3851,B 19.441,C -0.54,E1 19.3299,E2 227.4369} C_DIS
LIN {X -92.2044,Y -89.0944,Z 151,A -137.1435,B 19.4412,C -0.5336,E1 19.3342,E2 225.2019} C_DIS
LIN {X -86.0951,Y -95.011,Z 151,A -133.3246,B 19.4414,C -0.5265,E1 19.342,E2 221.3835} C_DIS
LIN {X -82.8337,Y -97.8678,Z 151,A -131.347,B 19.4414,C -0.5243,E1 19.3461,E2 219.4023} C_DIS
LIN {X -79.4813,Y -100.6097,Z 151,A -129.3657,B 19.4415,C -0.5225,E1 19.3505,E2 217.4167} C_DIS
LIN {X -75.5038,Y -103.6279,Z 151,A -127.1356,B 19.4416,C -0.5186,E1 19.3554,E2 215.1879} C_DIS
LIN {X -72.2515,Y -105.9212,Z 151,A -125.3359,B 19.4416,C -0.5166,E1 19.3596,E2 213.3865} C_DIS
LIN {X -68.9227,Y -108.1165,Z 151,A -123.5624,B 19.4418,C -0.5135,E1 19.3637,E2 211.6147} C_DIS
LIN {X -65.0659,Y -110.4804,Z 151,A -121.5367,B 19.4418,C -0.5107,E1 19.3686,E2 209.5891} C_DIS
LIN {X -61.0543,Y -112.7475,Z 151,A -119.4217,B 19.4418,C -0.51,E1 19.3738,E2 207.4682} C_DIS
LIN {X -57.2844,Y -114.7077,Z 151,A -117.6173,B 19.442,C -0.5041,E1 19.3782,E2 205.6753} C_DIS
LIN {X -54.063,Y -116.2593,Z 151,A -116.0143,B 19.442,C -0.5025,E1 19.3823,E2 204.0719} C_DIS
LIN {X -50.1467,Y -118.0039,Z 151,A -114.0774,B 19.442,C -0.5012,E1 19.3872,E2 202.1328} C_DIS
LIN {X -46.2299,Y -119.5903,Z 151,A -112.2229,B 19.4421,C -0.498,E1 19.392,E2 200.2825} C_DIS
LIN {X -42.5938,Y -120.9345,Z 151,A -110.4292,B 19.4421,C -0.4988,E1 19.3968,E2 198.4817} C_DIS
LIN {X -39.0061,Y -122.1373,Z 151,A -108.8473,B 19.4423,C -0.4933,E1 19.4009,E2 196.9125} C_DIS
LIN {X -35.8693,Y -123.0952,Z 151,A -107.316,B 19.4423,C -0.4948,E1 19.4051,E2 195.3734} C_DIS
LIN {X -32.2026,Y -124.1067,Z 151,A -105.5623,B 19.4423,C -0.4958,E1 19.4098,E2 193.6132} C_DIS
LIN {X -28.2634,Y -125.0612,Z 151,A -103.7505,B 19.4423,C -0.4949,E1 19.4147,E2 191.8011} C_DIS
LIN {X -24.04,Y -125.9409,Z 151,A -101.875,B 19.4423,C -0.492,E1 19.4199,E2 189.9313} C_DIS
LIN {X -19.9567,Y -126.6527,Z 151,A -100.0232,B 19.4423,C -0.4914,E1 19.425,E2 188.0792} C_DIS
LIN {X -14.5356,Y -127.39,Z 151,A -97.4748,B 19.4423,C -0.4949,E1 19.4321,E2 185.5179} C_DIS
LIN {X -8.5544,Y -127.9311,Z 151,A -94.988,B 19.4424,C -0.487,E1 19.4389,E2 183.0533} C_DIS
LIN {X -2.0501,Y -128.1987,Z 151,A -92.3534,B 19.4427,C -0.4764,E1 19.4462,E2 180.4498} C_DIS
LIN {X 0.9178,Y -128.1803,Z 151,A -90.7527,B 19.4424,C -0.4877,E1 19.4508,E2 178.8152} C_DIS
Enddeposition()
LIN {X 0.9178,Y -128.1803,Z 151,A -90.7527,B 19.4424,C -0.4877,E1 19.4508,E2 178.8152} C_DIS
Startdeposition()
$VEL.CP = VEL_PRINT
LIN {X -1.1917,Y -127.266,Z 151,A -92.0206,B 18.2102,C -0.3216,E1 18.2107,E2 180.486} C_DIS
LIN {X -5.603,Y -127.1488,Z 151,A -93.9068,B 18.2101,C -0.3251,E1 18.2054,E2 182.3615} C_DIS
LIN {X -9.3863,Y -126.924,Z 151,A -95.6149,B 18.2101,C -0.3251,E1 18.2007,E2 184.0705} C_DIS
LIN {X -13.2002,Y -126.5847,Z 151,A -97.4474,B 18.2101,C -0.3214,E1 18.1955,E2 185.916} C_DIS
LIN {X -17.1524,Y -126.1108,Z 151,A -99.1245,B 18.2101,C -0.3258,E1 18.1909,E2 187.5806} C_DIS
LIN {X -20.2359,Y -125.6534,Z 151,A -100.5527,B 18.2101,C -0.3253,E1 18.187,E2 189.012} C_DIS
LIN {X -23.3039,Y -125.1201,Z 151,A -101.9532,B 18.2101,C -0.3259,E1 18.1831,E2 190.4127} C_DIS
LIN {X -27.0622,Y -124.36,Z 151,A -103.6874,B 18.2101,C -0.3264,E1 18.1784,E2 192.1481} C_DIS
LIN {X -30.9267,Y -123.4561,Z 151,A -105.5355,B 18.2101,C -0.3253,E1 18.1733,E2 194.0035} C_DIS
LIN {X -34.9158,Y -122.3888,Z 151,A -107.4721,B 18.2101,C -0.3238,E1 18.1681,E2 195.9493} C_DIS
LIN {X -39.2379,Y -121.0718,Z 151,A -109.5281,B 18.2101,C -0.3245,E1 18.1626,E2 198.0078} C_DIS
LIN {X -43.4348,Y -119.6293,Z 151,A -111.3191,B 18.21,C -0.3335,E1 18.158,E2 199.7751} C_DIS
LIN {X -46.8378,Y -118.3406,Z 151,A -113.1512,B 18.21,C -0.3283,E1 18.1531,E2 201.6294} C_DIS
LIN {X -50.2651,Y -116.9237,Z 151,A -114.821,B 18.21,C -0.33,E1 18.1488,E2 203.299} C_DIS
LIN {X -53.7664,Y -115.3559,Z 151,A -116.4216,B 18.21,C -0.3363,E1 18.1448,E2 204.8849} C_DIS
LIN {X -56.5762,Y -114.0039,Z 151,A -117.9449,B 18.21,C -0.3339,E1 18.141,E2 206.4216} C_DIS
LIN {X -59.9884,Y -112.248,Z 151,A -119.7018,B 18.21,C -0.3351,E1 18.1366,E2 208.1815} C_DIS
LIN {X -63.4693,Y -110.3173,Z 151,A -121.5081,B 18.2099,C -0.3371,E1 18.1322,E2 209.9891} C_DIS
LIN {X -67.3881,Y -107.9677,Z 151,A -123.4466,B 18.2098,C -0.3441,E1 18.1276,E2 211.9134} C_DIS
LIN {X -70.1113,Y -106.2195,Z 151,A -124.8899,B 18.2098,C -0.3468,E1 18.1243,E2 213.3546} C_DIS
LIN {X -72.6898,Y -104.4717,Z 151,A -126.2959,B 18.2097,C -0.3489,E1 18.121,E2 214.7605} C_DIS
LIN {X -75.8056,Y -102.2337,Z 151,A -128.1266,B 18.2097,C -0.3483,E1 18.1169,E2 216.6022} C_DIS
LIN {X -78.9245,Y -99.846,Z 151,A -129.9104,B 18.2097,C -0.3509,E1 18.1129,E2 218.387} C_DIS
LIN {X -81.9457,Y -97.3812,Z 151,A -131.6542,B 18.2096,C -0.3545,E1 18.1092,E2 220.1285} C_DIS
LIN {X -85.1584,Y -94.5849,Z 151,A -133.6072,B 18.2096,C -0.357,E1 18.1051,E2 222.0845} C_DIS
LIN {X -88.0867,Y -91.8636,Z 151,A -135.375,B 18.2094,C -0.3617,E1 18.1015,E2 223.8476} C_DIS
LIN {X -91.0955,Y -88.8812,Z 151,A -137.3725,B 18.2094,C -0.3626,E1 18.0976,E2 225.8541} C_DIS
LIN {X -94.0649,Y -85.7322,Z 151,A -139.3344,B 18.2094,C -0.3664,E1 18.0938,E2 227.8162} C_DIS
LIN {X -96.8805,Y -82.5369,Z 151,A -141.205,B 18.2092,C -0.3722,E1 18.0904,E2 229.6801} C_DIS
LIN {X -99.3642,Y -79.53,Z 151,A -143.0467,B 18.2092,C -0.3733,E1 18.0872,E2 231.5301} C_DIS
LIN {X -102.2198,Y -75.8243,Z 151,A -145.0276,B 18.209,C -0.3824,E1 18.0838,E2 233.4952} C_DIS
LIN {X -104.4201,Y -72.7639,Z 151,A -146.5935,B 18.2088,C -0.3909,E1 18.0813,E2 235.0448} C_DIS
LIN {X -105.8281,Y -70.7006,Z 151,A -147.9937,B 18.209,C -0.3846,E1 18.0791,E2 236.4751} C_DIS
LIN {X -107.9755,Y -67.3755,Z 151,A -149.7848,B 18.2089,C -0.3888,E1 18.0764,E2 238.2656} C_DIS
LIN {X -110.3159,Y -63.4717,Z 151,A -151.729,B 18.2087,C -0.3975,E1 18.0737,E2 240.196} C_DIS
LIN {X -111.8939,Y -60.6467,Z 151,A -153.3493,B 18.2087,C -0.396,E1 18.0715,E2 241.8333} C_DIS
LIN {X -113.9597,Y -56.6657,Z 151,A -155.31,B 18.2086,C -0.4033,E1 18.069,E2 243.7854} C_DIS
LIN {X -115.7121,Y -52.9961,Z 151,A -157.0621,B 18.2084,C -0.4108,E1 18.067,E2 245.5266} C_DIS
LIN {X -116.9763,Y -50.1435,Z 151,A -158.6123,B 18.2084,C -0.41,E1 18.0652,E2 247.0917} C_DIS
LIN {X -118.7437,Y -45.8009,Z 151,A -160.732,B 18.2084,C -0.4156,E1 18.063,E2 249.21} C_DIS
LIN {X -120.3457,Y -41.4089,Z 151,A -162.724,B 18.2081,C -0.4253,E1 18.0612,E2 251.187} C_DIS
LIN {X -121.3676,Y -38.3119,Z 151,A -164.3547,B 18.2081,C -0.4243,E1 18.0598,E2 252.8342} C_DIS
LIN {X -122.6607,Y -33.9437,Z 151,A -166.2708,B 18.2079,C -0.4346,E1 18.0583,E2 254.7326} C_DIS
LIN {X -123.4565,Y -30.9251,Z 151,A -167.6869,B 18.2079,C -0.4384,E1 18.0573,E2 256.1482} C_DIS
LIN {X -124.2407,Y -27.6141,Z 151,A -169.401,B 18.2079,C -0.4371,E1 18.0562,E2 257.8809} C_DIS
LIN {X -124.9876,Y -23.9966,Z 151,A -170.9135,B 18.2076,C -0.4469,E1 18.0554,E2 259.3744} C_DIS
LIN {X -125.5381,Y -20.9271,Z 151,A -172.2834,B 18.2075,C -0.4523,E1 18.0548,E2 260.7386} C_DIS
LIN {X -125.9961,Y -17.9652,Z 151,A -173.7117,B 18.2075,C -0.4538,E1 18.0542,E2 262.1741} C_DIS
LIN {X -126.4968,Y -14.0175,Z 151,A -175.506,B 18.2073,C -0.4592,E1 18.0536,E2 263.9663} C_DIS
LIN {X -126.8018,Y -10.9146,Z 151,A -176.9175,B 18.2073,C -0.4632,E1 18.0532,E2 265.3767} C_DIS
LIN {X -127.031,Y -7.8041,Z 151,A -178.3276,B 18.2071,C -0.4673,E1 18.0529,E2 266.7856} C_DIS
LIN {X -127.1996,Y -4.3003,Z 151,A 179.9444,B 18.2071,C -0.4673,E1 18.0527,E2 268.5282} C_DIS
LIN {X -127.274,Y -0.017,Z 151,A 178.0591,B 18.2069,C -0.4747,E1 18.0527,E2 270.406} C_DIS
LIN {X -127.2335,Y 3.1031,Z 151,A 176.5474,B 18.2069,C -0.4757,E1 18.0527,E2 271.9276} C_DIS
LIN {X -127.0753,Y 7.0799,Z 151,A 174.7568,B 18.2068,C -0.4812,E1 18.053,E2 273.7155} C_DIS
LIN {X -126.8013,Y 10.9203,Z 151,A 173.1264,B 18.2065,C -0.4899,E1 18.0534,E2 275.3319} C_DIS
LIN {X -126.3989,Y 14.8702,Z 151,A 171.2339,B 18.2065,C -0.492,E1 18.054,E2 277.2336} C_DIS
LIN {X -125.8948,Y 18.6739,Z 151,A 169.6288,B 18.2062,C -0.5012,E1 18.0546,E2 278.8226} C_DIS
LIN {X -125.3994,Y 21.7529,Z 151,A 168.1831,B 18.2062,C -0.5042,E1 18.0552,E2 280.2709} C_DIS
LIN {X -124.8281,Y 24.8194,Z 151,A 166.6012,B 18.2062,C -0.5028,E1 18.0561,E2 281.8706} C_DIS
LIN {X -123.991,Y 28.707,Z 151,A 164.9735,B 18.2059,C -0.5135,E1 18.0571,E2 283.4774} C_DIS
LIN {X -123.2159,Y 31.8731,Z 151,A 163.3358,B 18.2059,C -0.5125,E1 18.0582,E2 285.132} C_DIS
LIN {X -122.0199,Y 36.1806,Z 151,A 161.4285,B 18.2057,C -0.5219,E1 18.0596,E2 287.0245} C_DIS
LIN {X -120.8464,Y 39.9241,Z 151,A 159.5986,B 18.2056,C -0.5251,E1 18.0612,E2 288.859} C_DIS
LIN {X -119.5414,Y 43.6789,Z 151,A 157.8713,B 18.2054,C -0.5324,E1 18.0628,E2 290.5767} C_DIS
LIN {X -118.1706,Y 47.2599,Z 151,A 156.1337,B 18.2052,C -0.5371,E1 18.0646,E2 292.3129} C_DIS
LIN {X -116.6907,Y 50.8041,Z 151,A 154.3644,B 18.2052,C -0.5408,E1 18.0665,E2 294.0842} C_DIS
LIN {X -115.3345,Y 53.8126,Z 151,A 152.8873,B 18.205,C -0.5453,E1 18.0682,E2 295.5582} C_DIS
LIN {X -113.9907,Y 56.6028,Z 151,A 151.3647,B 18.205,C -0.5452,E1 18.0701,E2 297.093} C_DIS
LIN {X -112.2421,Y 59.9994,Z 151,A 149.6136,B 18.205,C -0.5489,E1 18.0724,E2 298.8451} C_DIS
LIN {X -110.3322,Y 63.4436,Z 151,A 147.8082,B 18.2048,C -0.5528,E1 18.0749,E2 300.6516} C_DIS
LIN {X -108.3542,Y 66.7651,Z 151,A 146.2061,B 18.2045,C -0.562,E1 18.0772,E2 302.2358} C_DIS
LIN {X -106.6858,Y 69.3996,Z 151,A 144.6841,B 18.2045,C -0.5619,E1 18.0795,E2 303.7689} C_DIS
LIN {X -104.4481,Y 72.7238,Z 151,A 142.9795,B 18.2043,C -0.5698,E1 18.0821,E2 305.4599} C_DIS
LIN {X -102.6461,Y 75.2458,Z 151,A 141.4351,B 18.2043,C -0.5686,E1 18.0847,E2 307.0189} C_DIS
LIN {X -99.8492,Y 78.9205,Z 151,A 139.377,B 18.2041,C -0.5745,E1 18.0882,E2 309.0718} C_DIS
LIN {X -97.3848,Y 81.9413,Z 151,A 137.6306,B 18.2041,C -0.5791,E1 18.0913,E2 310.8148} C_DIS
LIN {X -94.59,Y 85.1527,Z 151,A 135.6584,B 18.2039,C -0.5819,E1 18.095,E2 312.7906} C_DIS
LIN {X -91.6316,Y 88.3283,Z 151,A 133.6615,B 18.2039,C -0.5851,E1 18.0988,E2 314.7896} C_DIS
LIN {X -88.583,Y 91.3849,Z 151,A 131.7865,B 18.2036,C -0.5917,E1 18.1025,E2 316.6544} C_DIS
LIN {X -85.7444,Y 94.0539,Z 151,A 129.9429,B 18.2036,C -0.5926,E1 18.1063,E2 318.5057} C_DIS
LIN {X -82.5326,Y 96.8841,Z 151,A 128.0687,B 18.2034,C -0.5985,E1 18.1102,E2 320.3714} C_DIS
LIN {X -79.5275,Y 99.3662,Z 151,A 126.3297,B 18.2033,C -0.6026,E1 18.114,E2 322.1066} C_DIS
LIN {X -76.3976,Y 101.7923,Z 151,A 124.4625,B 18.2033,C -0.6033,E1 18.1182,E2 323.9809} C_DIS
LIN {X -73.2804,Y 104.0583,Z 151,A 122.8477,B 18.203,C -0.6106,E1 18.1218,E2 325.5803} C_DIS
LIN {X -70.7079,Y 105.8232,Z 151,A 121.3602,B 18.203,C -0.6104,E1 18.1252,E2 327.0754} C_DIS
LIN {X -67.3636,Y 107.983,Z 151,A 119.4977,B 18.203,C -0.6112,E1 18.1297,E2 328.9437} C_DIS
LIN {X -63.4654,Y 110.3196,Z 151,A 117.5612,B 18.2028,C -0.6183,E1 18.1343,E2 330.8656} C_DIS
LIN {X -60.6442,Y 111.8953,Z 151,A 116.0405,B 18.2028,C -0.6184,E1 18.138,E2 332.3921} C_DIS
LIN {X -57.9521,Y 113.3105,Z 151,A 114.6643,B 18.2027,C -0.6203,E1 18.1414,E2 333.7675} C_DIS
LIN {X -54.4015,Y 115.0583,Z 151,A 112.949,B 18.2025,C -0.6252,E1 18.1457,E2 335.4736} C_DIS
LIN {X -51.5677,Y 116.3556,Z 151,A 111.5418,B 18.2025,C -0.627,E1 18.1493,E2 336.8799} C_DIS
LIN {X -48.0365,Y 117.8576,Z 151,A 109.6292,B 18.2026,C -0.623,E1 18.1543,E2 338.8113} C_DIS
LIN {X -43.6777,Y 119.5418,Z 151,A 107.6623,B 18.2024,C -0.6301,E1 18.1594,E2 340.7611} C_DIS
LIN {X -40.4219,Y 120.6806,Z 151,A 106.0388,B 18.2024,C -0.6295,E1 18.1637,E2 342.3909} C_DIS
LIN {X -36.2375,Y 122.0032,Z 151,A 103.9804,B 18.2024,C -0.6287,E1 18.1692,E2 344.4568} C_DIS
LIN {X -32.4284,Y 123.0701,Z 151,A 102.3774,B 18.2022,C -0.6364,E1 18.1735,E2 346.0386} C_DIS
LIN {X -28.7009,Y 123.9924,Z 151,A 100.606,B 18.2022,C -0.6364,E1 18.1783,E2 347.8134} C_DIS
LIN {X -25.5793,Y 124.6735,Z 151,A 99.178,B 18.2022,C -0.6379,E1 18.1822,E2 349.2391} C_DIS
LIN {X -22.4341,Y 125.2775,Z 151,A 97.7569,B 18.202,C -0.6396,E1 18.1861,E2 350.6568} C_DIS
LIN {X -19.4867,Y 125.7697,Z 151,A 96.4091,B 18.202,C -0.6403,E1 18.1898,E2 352.0039} C_DIS
LIN {X -16.2858,Y 126.2244,Z 151,A 94.815,B 18.2022,C -0.6363,E1 18.1942,E2 353.6126} C_DIS
LIN {X -12.4585,Y 126.6596,Z 151,A 93.071,B 18.2022,C -0.6368,E1 18.1991,E2 355.3566} C_DIS
LIN {X -8.6386,Y 126.9786,Z 151,A 91.4859,B 18.202,C -0.6423,E1 18.2034,E2 356.925} C_DIS
LIN {X -5.5023,Y 127.1527,Z 151,A 90.0227,B 18.202,C -0.6409,E1 18.2075,E2 358.3929} C_DIS
LIN {X -2.2755,Y 127.2503,Z 151,A 88.5302,B 18.202,C -0.6399,E1 18.2117,E2 359.889} C_DIS
LIN {X 1.5998,Y 127.2616,Z 151,A 86.8555,B 18.202,C -0.6425,E1 18.2164,E2 361.5551} C_DIS
LIN {X 4.7065,Y 127.1838,Z 151,A 85.4657,B 18.202,C -0.6429,E1 18.2202,E2 362.9432} C_DIS
LIN {X 7.815,Y 127.0304,Z 151,A 84.0133,B 18.202,C -0.641,E1 18.2243,E2 364.4008} C_DIS
LIN {X 11.7571,Y 126.7269,Z 151,A 82.3077,B 18.202,C -0.6434,E1 18.229,E2 366.0974} C_DIS
LIN {X 14.886,Y 126.397,Z 151,A 80.9019,B 18.202,C -0.6435,E1 18.2329,E2 367.5015} C_DIS
LIN {X 17.9761,Y 125.9945,Z 151,A 79.4739,B 18.202,C -0.6422,E1 18.2369,E2 368.932} C_DIS
LIN {X 20.9352,Y 125.5367,Z 151,A 78.1274,B 18.202,C -0.6418,E1 18.2406,E2 370.278} C_DIS
LIN {X 24.0024,Y 124.9865,Z 151,A 76.649,B 18.202,C -0.6385,E1 18.2447,E2 371.7645} C_DIS
LIN {X 27.8878,Y 124.1781,Z 151,A 74.8746,B 18.2021,C -0.638,E1 18.2495,E2 373.5373} C_DIS
LIN {X 31.745,Y 123.2484,Z 151,A 73.1617,B 18.2021,C -0.6395,E1 18.2541,E2 375.2417} C_DIS
LIN {X 35.4476,Y 122.2345,Z 151,A 71.4328,B 18.2021,C -0.6382,E1 18.2588,E2 376.9704} C_DIS
LIN {X 38.4341,Y 121.3285,Z 151,A 70.0312,B 18.2021,C -0.6372,E1 18.2625,E2 378.3717} C_DIS
LIN {X 41.5817,Y 120.2858,Z 151,A 68.433,B 18.2023,C -0.6322,E1 18.2668,E2 379.9816} C_DIS
LIN {X 45.1445,Y 118.9955,Z 151,A 66.6839,B 18.2024,C -0.6289,E1 18.2714,E2 381.7358} C_DIS
LIN {X 48.7098,Y 117.5804,Z 151,A 64.9725,B 18.2024,C -0.6277,E1 18.2758,E2 383.4454} C_DIS
LIN {X 52.3445,Y 116.0082,Z 151,A 63.3393,B 18.2024,C -0.6311,E1 18.2799,E2 385.0621} C_DIS
LIN {X 55.1703,Y 114.6909,Z 151,A 61.939,B 18.2024,C -0.6296,E1 18.2834,E2 386.4622} C_DIS
LIN {X 58.6153,Y 112.9703,Z 151,A 60.2408,B 18.2024,C -0.6286,E1 18.2877,E2 388.1568} C_DIS
LIN {X 62.026,Y 111.1354,Z 151,A 58.4522,B 18.2026,C -0.6246,E1 18.2921,E2 389.951} C_DIS
LIN {X 65.44,Y 109.1598,Z 151,A 56.5607,B 18.2028,C -0.6178,E1 18.2966,E2 391.856} C_DIS
LIN {X 68.799,Y 107.0742,Z 151,A 54.9371,B 18.2027,C -0.6208,E1 18.3004,E2 393.4626} C_DIS
LIN {X 71.3967,Y 105.3597,Z 151,A 53.3979,B 18.2029,C -0.6134,E1 18.3041,E2 395.0179} C_DIS
LIN {X 74.8813,Y 102.9126,Z 151,A 51.546,B 18.2029,C -0.6126,E1 18.3082,E2 396.8632} C_DIS
LIN {X 78.3096,Y 100.329,Z 151,A 49.6149,B 18.2031,C -0.6092,E1 18.3125,E2 398.7951} C_DIS
LIN {X 81.3454,Y 97.8833,Z 151,A 47.8787,B 18.2031,C -0.6067,E1 18.3163,E2 400.53} C_DIS
LIN {X 84.6194,Y 95.0677,Z 151,A 45.873,B 18.2033,C -0.6006,E1 18.3205,E2 402.5438} C_DIS
LIN {X 87.753,Y 92.1826,Z 151,A 44.0497,B 18.2033,C -0.6003,E1 18.3242,E2 404.3575} C_DIS
LIN {X 90.5547,Y 89.4323,Z 151,A 42.2079,B 18.2035,C -0.5938,E1 18.3279,E2 406.209} C_DIS
LIN {X 93.4952,Y 86.3533,Z 151,A 40.3156,B 18.2036,C -0.5906,E1 18.3315,E2 408.0998} C_DIS
LIN {X 96.3707,Y 83.1315,Z 151,A 38.465,B 18.2036,C -0.5898,E1 18.3349,E2 409.9412} C_DIS
LIN {X 98.8718,Y 80.1411,Z 151,A 36.6377,B 18.2039,C -0.583,E1 18.3381,E2 411.7781} C_DIS
LIN {X 101.7219,Y 76.4909,Z 151,A 34.6842,B 18.2039,C -0.583,E1 18.3414,E2 413.7183} C_DIS
LIN {X 104.0694,Y 73.2647,Z 151,A 32.9363,B 18.2039,C -0.5805,E1 18.3443,E2 415.4623} C_DIS
LIN {X 105.8284,Y 70.7001,Z 151,A 31.4806,B 18.2041,C -0.5749,E1 18.3466,E2 416.9256} C_DIS
LIN {X 107.9702,Y 67.384,Z 151,A 29.7873,B 18.2041,C -0.5736,E1 18.3491,E2 418.6109} C_DIS
LIN {X 109.5973,Y 64.7044,Z 151,A 28.243,B 18.2044,C -0.5649,E1 18.3513,E2 420.1717} C_DIS
LIN {X 111.4994,Y 61.369,Z 151,A 26.5316,B 18.2046,C -0.561,E1 18.3537,E2 421.8829} C_DIS
LIN {X 113.3627,Y 57.8495,Z 151,A 24.9211,B 18.2045,C -0.5632,E1 18.3557,E2 423.4743} C_DIS
LIN {X 114.8727,Y 54.79,Z 151,A 23.2994,B 18.2047,C -0.5558,E1 18.3577,E2 425.1075} C_DIS
LIN {X 116.3519,Y 51.576,Z 151,A 21.7551,B 18.2047,C -0.5532,E1 18.3595,E2 426.648} C_DIS
LIN {X 117.8949,Y 47.9438,Z 151,A 19.8693,B 18.205,C -0.5441,E1 18.3615,E2 428.5481} C_DIS
LIN {X 119.5451,Y 43.6686,Z 151,A 17.7881,B 18.2052,C -0.5375,E1 18.3636,E2 430.6339} C_DIS
LIN {X 120.8268,Y 39.983,Z 151,A 16.1905,B 18.2052,C -0.5386,E1 18.365,E2 432.2153} C_DIS
LIN {X 122.0331,Y 36.1354,Z 151,A 14.2838,B 18.2055,C -0.5297,E1 18.3665,E2 434.1346} C_DIS
LIN {X 123.0674,Y 32.4386,Z 151,A 12.7196,B 18.2055,C -0.531,E1 18.3677,E2 435.6822} C_DIS
LIN {X 123.9917,Y 28.704,Z 151,A 10.9586,B 18.2055,C -0.5247,E1 18.3688,E2 437.4486} C_DIS
LIN {X 124.8282,Y 24.8189,Z 151,A 9.234,B 18.2057,C -0.5218,E1 18.3698,E2 439.1682} C_DIS
LIN {X 125.3986,Y 21.7576,Z 151,A 7.7574,B 18.2059,C -0.5147,E1 18.3706,E2 440.6551} C_DIS
LIN {X 126.0115,Y 17.8568,Z 151,A 6.0645,B 18.2059,C -0.5126,E1 18.3713,E2 442.3407} C_DIS
LIN {X 126.4994,Y 13.9934,Z 151,A 4.3304,B 18.2061,C -0.508,E1 18.3718,E2 444.0749} C_DIS
LIN {X 126.8732,Y 10.0689,Z 151,A 2.5993,B 18.2061,C -0.5042,E1 18.3723,E2 445.8035} C_DIS
LIN {X 127.0821,Y 6.9446,Z 151,A 1.1756,B 18.2063,C -0.4994,E1 18.3725,E2 447.2306} C_DIS
LIN {X 127.2149,Y 3.7728,Z 151,A -0.2396,B 18.2063,C -0.4955,E1 18.3726,E2 448.6462} C_DIS
LIN {X 127.274,Y -0.0287,Z 151,A -2.0051,B 18.2066,C -0.4881,E1 18.3726,E2 450.4204} C_DIS
LIN {X 127.2328,Y -3.1277,Z 151,A -3.3283,B 18.2066,C -0.4866,E1 18.3726,E2 451.7372} C_DIS
LIN {X 127.1161,Y -6.2682,Z 151,A -4.721,B 18.2067,C -0.4831,E1 18.3725,E2 453.1293} C_DIS
LIN {X 126.9252,Y -9.3694,Z 151,A -6.1305,B 18.2068,C -0.4783,E1 18.3722,E2 454.5421} C_DIS
LIN {X 126.583,Y -13.216,Z 151,A -7.8676,B 18.207,C -0.473,E1 18.3717,E2 456.2815} C_DIS
LIN {X 126.2225,Y -16.3003,Z 151,A -9.2881,B 18.207,C -0.4678,E1 18.3712,E2 457.7067} C_DIS
LIN {X 125.6584,Y -20.2055,Z 151,A -10.9977,B 18.2072,C -0.4649,E1 18.3705,E2 459.4112} C_DIS
LIN {X 125.1196,Y -23.3063,Z 151,A -12.3887,B 18.2072,C -0.4616,E1 18.3698,E2 460.8013} C_DIS
LIN {X 124.3588,Y -27.0679,Z 151,A -14.1067,B 18.2074,C -0.4567,E1 18.3689,E2 462.5207} C_DIS
LIN {X 123.6301,Y -30.224,Z 151,A -15.5361,B 18.2074,C -0.4534,E1 18.3679,E2 463.9489} C_DIS
LIN {X 122.6621,Y -33.9387,Z 151,A -17.4121,B 18.2077,C -0.4424,E1 18.3666,E2 465.8445} C_DIS
LIN {X 121.3277,Y -38.4368,Z 151,A -19.4527,B 18.2077,C -0.4388,E1 18.3649,E2 467.88} C_DIS
LIN {X 120.1017,Y -42.1127,Z 151,A -21.0871,B 18.2078,C -0.4379,E1 18.3634,E2 469.5043} C_DIS
LIN {X 118.9934,Y -45.1503,Z 151,A -22.6783,B 18.208,C -0.4283,E1 18.3619,E2 471.1134} C_DIS
LIN {X 117.581,Y -48.7084,Z 151,A -24.3755,B 18.2081,C -0.4243,E1 18.3601,E2 472.81} C_DIS
LIN {X 116.0106,Y -52.3389,Z 151,A -25.9987,B 18.2081,C -0.4252,E1 18.3583,E2 474.4177} C_DIS
LIN {X 114.695,Y -55.1618,Z 151,A -27.4289,B 18.2082,C -0.4201,E1 18.3566,E2 475.8532} C_DIS
LIN {X 112.9726,Y -58.6109,Z 151,A -29.0834,B 18.2082,C -0.4184,E1 18.3545,E2 477.501} C_DIS
LIN {X 111.3942,Y -61.5589,Z 151,A -30.7259,B 18.2085,C -0.4088,E1 18.3523,E2 479.1616} C_DIS
LIN {X 109.159,Y -65.4414,Z 151,A -32.7508,B 18.2085,C -0.403,E1 18.3494,E2 481.1903} C_DIS
LIN {X 107.0682,Y -68.8084,Z 151,A -34.52,B 18.2087,C -0.3987,E1 18.3467,E2 482.9604} C_DIS
LIN {X 104.8318,Y -72.1698,Z 151,A -36.3065,B 18.2087,C -0.3951,E1 18.3439,E2 484.7459} C_DIS
LIN {X 102.6577,Y -75.2301,Z 151,A -37.9998,B 18.2089,C -0.3906,E1 18.3412,E2 486.442} C_DIS
LIN {X 99.8419,Y -78.9298,Z 151,A -40.0942,B 18.2089,C -0.3852,E1 18.3376,E2 488.5395} C_DIS
LIN {X 96.9965,Y -82.4004,Z 151,A -42.0455,B 18.209,C -0.3828,E1 18.3341,E2 490.4857} C_DIS
LIN {X 94.2539,Y -85.5239,Z 151,A -43.8672,B 18.209,C -0.3802,E1 18.3307,E2 492.3042} C_DIS
LIN {X 91.6129,Y -88.3475,Z 151,A -45.6709,B 18.2092,C -0.3737,E1 18.3272,E2 494.1175} C_DIS
LIN {X 88.5787,Y -91.3891,Z 151,A -47.5134,B 18.2092,C -0.3727,E1 18.3236,E2 495.9521} C_DIS
LIN {X 85.6912,Y -94.1021,Z 151,A -49.3514,B 18.2093,C -0.3667,E1 18.3198,E2 497.7987} C_DIS
LIN {X 82.517,Y -96.8974,Z 151,A -51.1908,B 18.2093,C -0.365,E1 18.3159,E2 499.6331} C_DIS
LIN {X 79.5212,Y -99.3712,Z 151,A -53.0038,B 18.2095,C -0.359,E1 18.312,E2 501.4557} C_DIS
LIN {X 76.2324,Y -101.9159,Z 151,A -54.824,B 18.2095,C -0.3572,E1 18.3079,E2 503.2723} C_DIS
LIN {X 73.2717,Y -104.0645,Z 151,A -56.3499,B 18.2095,C -0.3585,E1 18.3045,E2 504.7862} C_DIS
LIN {X 70.7203,Y -105.8149,Z 151,A -57.7374,B 18.2095,C -0.3561,E1 18.3013,E2 506.1747} C_DIS
LIN {X 67.54,Y -107.8732,Z 151,A -59.4768,B 18.2096,C -0.3517,E1 18.2972,E2 507.92} C_DIS
LIN {X 64.0288,Y -109.9934,Z 151,A -61.2757,B 18.2096,C -0.3503,E1 18.2929,E2 509.7155} C_DIS
LIN {X 60.6259,Y -111.9053,Z 151,A -63.0985,B 18.2097,C -0.345,E1 18.2884,E2 511.5479} C_DIS
LIN {X 57.8633,Y -113.3557,Z 151,A -64.4465,B 18.2097,C -0.345,E1 18.2851,E2 512.8908} C_DIS
LIN {X 54.4099,Y -115.0542,Z 151,A -66.149,B 18.2097,C -0.3434,E1 18.2808,E2 514.5916} C_DIS
LIN {X 51.5428,Y -116.3667,Z 151,A -67.5574,B 18.2098,C -0.3418,E1 18.2772,E2 516.0002} C_DIS
LIN {X 48.0197,Y -117.8644,Z 151,A -69.447,B 18.21,C -0.3333,E1 18.2723,E2 517.9108} C_DIS
LIN {X 44.3463,Y -119.2945,Z 151,A -71.0399,B 18.2099,C -0.3378,E1 18.2682,E2 519.4844} C_DIS
LIN {X 41.3972,Y -120.3497,Z 151,A -72.5741,B 18.2099,C -0.3315,E1 18.2641,E2 521.0342} C_DIS
LIN {X 37.6307,Y -121.5804,Z 151,A -74.2241,B 18.2099,C -0.3345,E1 18.2597,E2 522.6704} C_DIS
LIN {X 34.3527,Y -122.5463,Z 151,A -75.8321,B 18.21,C -0.3303,E1 18.2554,E2 524.2877} C_DIS
LIN {X 30.9086,Y -123.4607,Z 151,A -77.5054,B 18.21,C -0.3263,E1 18.2508,E2 525.9704} C_DIS
LIN {X 27.0536,Y -124.3619,Z 151,A -79.1364,B 18.21,C -0.3303,E1 18.2464,E2 527.5853} C_DIS
LIN {X 24.0014,Y -124.9867,Z 151,A -80.5349,B 18.21,C -0.3294,E1 18.2426,E2 528.9844} C_DIS
LIN {X 20.807,Y -125.5581,Z 151,A -81.965,B 18.21,C -0.3294,E1 18.2387,E2 530.412} C_DIS
LIN {X 17.8929,Y -126.0064,Z 151,A -83.329,B 18.21,C -0.3273,E1 18.2349,E2 531.7811} C_DIS
LIN {X 14.0098,Y -126.4976,Z 151,A -85.2182,B 18.2102,C -0.3217,E1 18.2296,E2 533.6862} C_DIS
LIN {X 9.9984,Y -126.8792,Z 151,A -86.8657,B 18.2101,C -0.3269,E1 18.2251,E2 535.3156} C_DIS
LIN {X 7.0533,Y -127.0767,Z 151,A -88.2294,B 18.2101,C -0.3252,E1 18.2213,E2 536.6842} C_DIS
LIN {X 3.7847,Y -127.2145,Z 151,A -89.69,B 18.2101,C -0.3252,E1 18.2172,E2 538.144} C_DIS
LIN {X 0.9073,Y -127.2663,Z 151,A -90.4427,B 18.2098,C -0.3446,E1 18.2153,E2 538.8345} C_DIS
Enddeposition()
LIN {X 0.9471,Y -134.1856,Z 152,A -92.9033,B 24.9694,C -1.2773,E1 25.0007,E2 539.5173} C_DIS
Startdeposition()
$VEL.CP = VEL_PRINT
LIN {X 4.8031,Y -134.1048,Z 152,A -90.5794,B 24.9677,C -1.3138,E1 25.0074,E2 537.1072} C_DIS
LIN {X 9.0907,Y -133.8835,Z 152,A -88.7685,B 24.9677,C -1.3134,E1 25.0124,E2 535.298} C_DIS
LIN {X 12.5374,Y -133.6033,Z 152,A -87.3299,B 24.9677,C -1.3122,E1 25.0164,E2 533.8631} C_DIS
LIN {X 16.5009,Y -133.1729,Z 152,A -85.6328,B 24.9677,C -1.3129,E1 25.0211,E2 532.1655} C_DIS
LIN {X 20.3842,Y -132.6327,Z 152,A -84.0328,B 24.9679,C -1.3101,E1 25.0255,E2 530.5735} C_DIS
LIN {X 23.2207,Y -132.1662,Z 152,A -82.6952,B 24.9675,C -1.3171,E1 25.0293,E2 529.2209} C_DIS
LIN {X 27.0716,Y -131.4311,Z 152,A -81.0142,B 24.9675,C -1.3189,E1 25.0339,E2 527.5376} C_DIS
LIN {X 31.2779,Y -130.4937,Z 152,A -79.2637,B 24.9675,C -1.3158,E1 25.0386,E2 525.7968} C_DIS
LIN {X 34.1527,Y -129.7716,Z 152,A -77.9524,B 24.9674,C -1.3197,E1 25.0422,E2 524.4785} C_DIS
LIN {X 37.6576,Y -128.7974,Z 152,A -76.5318,B 24.9677,C -1.3142,E1 25.0459,E2 523.0732} C_DIS
LIN {X 40.6444,Y -127.8864,Z 152,A -75.2028,B 24.9676,C -1.3156,E1 25.0495,E2 521.7434} C_DIS
LIN {X 44.0167,Y -126.7651,Z 152,A -73.6212,B 24.9673,C -1.321,E1 25.0537,E2 520.1519} C_DIS
LIN {X 47.5653,Y -125.4778,Z 152,A -72.0017,B 24.9672,C -1.3236,E1 25.0579,E2 518.5296} C_DIS
LIN {X 51.2693,Y -124.0102,Z 152,A -70.2634,B 24.967,C -1.3282,E1 25.0625,E2 516.7846} C_DIS
LIN {X 54.7214,Y -122.5251,Z 152,A -68.7447,B 24.967,C -1.3259,E1 25.0663,E2 515.2748} C_DIS
LIN {X 57.5115,Y -121.2411,Z 152,A -67.3573,B 24.9668,C -1.3322,E1 25.0699,E2 513.8762} C_DIS
LIN {X 60.5811,Y -119.7366,Z 152,A -65.8931,B 24.9666,C -1.3349,E1 25.0735,E2 512.4095} C_DIS
LIN {X 63.9062,Y -117.9979,Z 152,A -64.2895,B 24.9665,C -1.3378,E1 25.0775,E2 510.8037} C_DIS
LIN {X 67.6332,Y -115.9019,Z 152,A -62.4273,B 24.9662,C -1.3432,E1 25.082,E2 508.9344} C_DIS
LIN {X 71.1948,Y -113.7487,Z 152,A -60.6612,B 24.9661,C -1.346,E1 25.0862,E2 507.1671} C_DIS
LIN {X 74.833,Y -111.3891,Z 152,A -58.8325,B 24.9659,C -1.3485,E1 25.0905,E2 505.3386} C_DIS
LIN {X 78.3083,Y -108.9737,Z 152,A -57.051,B 24.9659,C -1.3509,E1 25.0945,E2 503.5577} C_DIS
LIN {X 81.4669,Y -106.6325,Z 152,A -55.3942,B 24.9657,C -1.3533,E1 25.0982,E2 501.9011} C_DIS
LIN {X 84.8177,Y -103.9871,Z 152,A -53.5778,B 24.9655,C -1.3571,E1 25.1022,E2 500.0827} C_DIS
LIN {X 87.793,Y -101.488,Z 152,A -51.9169,B 24.9653,C -1.361,E1 25.1057,E2 498.4189} C_DIS
LIN {X 90.7483,Y -98.8539,Z 152,A -50.2287,B 24.9651,C -1.365,E1 25.1092,E2 496.7282} C_DIS
LIN {X 93.9863,Y -95.7806,Z 152,A -48.378,B 24.9651,C -1.3666,E1 25.1129,E2 494.8815} C_DIS
LIN {X 96.6392,Y -93.1038,Z 152,A -46.7229,B 24.9647,C -1.3732,E1 25.1162,E2 493.2178} C_DIS
LIN {X 99.3627,Y -90.1909,Z 152,A -45.0588,B 24.9646,C -1.3755,E1 25.1193,E2 491.5557} C_DIS
LIN {X 101.9351,Y -87.2739,Z 152,A -43.3918,B 24.9643,C -1.3802,E1 25.1224,E2 489.8849} C_DIS
LIN {X 104.6436,Y -84.0069,Z 152,A -41.6201,B 24.9642,C -1.3829,E1 25.1255,E2 488.1152} C_DIS
LIN {X 107.2841,Y -80.6074,Z 152,A -39.7323,B 24.9638,C -1.3908,E1 25.1287,E2 486.2178} C_DIS
LIN {X 109.9307,Y -76.9593,Z 152,A -37.7908,B 24.9634,C -1.3972,E1 25.1319,E2 484.2706} C_DIS
LIN {X 112.483,Y -73.1774,Z 152,A -35.9132,B 24.9634,C -1.3989,E1 25.1347,E2 482.3985} C_DIS
LIN {X 114.6948,Y -69.6601,Z 152,A -34.107,B 24.963,C -1.4059,E1 25.1374,E2 480.5848} C_DIS
LIN {X 116.9372,Y -65.8259,Z 152,A -32.2381,B 24.9628,C -1.41,E1 25.14,E2 478.7159} C_DIS
LIN {X 119.1909,Y -61.6525,Z 152,A -30.2643,B 24.9626,C -1.4132,E1 25.1426,E2 476.7449} C_DIS
LIN {X 120.9361,Y -58.1498,Z 152,A -28.6083,B 24.9624,C -1.4176,E1 25.1446,E2 475.0876} C_DIS
LIN {X 122.4198,Y -54.9568,Z 152,A -27.1455,B 24.9622,C -1.4199,E1 25.1463,E2 473.6271} C_DIS
LIN {X 123.7454,Y -51.9034,Z 152,A -25.807,B 24.9622,C -1.4197,E1 25.1478,E2 472.2964} C_DIS
LIN {X 125.0248,Y -48.7407,Z 152,A -24.3356,B 24.962,C -1.4252,E1 25.1493,E2 470.8203} C_DIS
LIN {X 126.1825,Y -45.6602,Z 152,A -22.9213,B 24.9617,C -1.4302,E1 25.1506,E2 469.4021} C_DIS
LIN {X 127.8087,Y -40.8877,Z 152,A -20.7655,B 24.9613,C -1.4372,E1 25.1526,E2 467.2419} C_DIS
LIN {X 128.8407,Y -37.51,Z 152,A -19.2485,B 24.961,C -1.4426,E1 25.1538,E2 465.7209} C_DIS
LIN {X 129.8669,Y -33.7949,Z 152,A -17.5984,B 24.9607,C -1.4482,E1 25.155,E2 464.0671} C_DIS
LIN {X 130.7682,Y -30.1103,Z 152,A -15.9904,B 24.9605,C -1.4529,E1 25.156,E2 462.4574} C_DIS
LIN {X 131.5714,Y -26.3822,Z 152,A -14.4143,B 24.9603,C -1.4553,E1 25.1569,E2 460.8849} C_DIS
LIN {X 132.2705,Y -22.6213,Z 152,A -12.7011,B 24.9598,C -1.4652,E1 25.1577,E2 459.1583} C_DIS
LIN {X 132.828,Y -19.07,Z 152,A -11.3562,B 24.9601,C -1.4595,E1 25.1583,E2 457.8347} C_DIS
LIN {X 133.2035,Y -16.2446,Z 152,A -10.0107,B 24.9595,C -1.4708,E1 25.1588,E2 456.4705} C_DIS
LIN {X 133.6513,Y -12.0349,Z 152,A -8.1707,B 24.959,C -1.4786,E1 25.1593,E2 454.623} C_DIS
LIN {X 133.9195,Y -8.5204,Z 152,A -6.73,B 24.959,C -1.48,E1 25.1595,E2 453.1875} C_DIS
LIN {X 134.1167,Y -4.496,Z 152,A -4.9832,B 24.9586,C -1.4872,E1 25.1597,E2 451.4343} C_DIS
LIN {X 134.1914,Y -0.3706,Z 152,A -3.1692,B 24.9581,C -1.496,E1 25.1597,E2 449.6103} C_DIS
LIN {X 134.1437,Y 3.5335,Z 152,A -1.6673,B 24.9583,C -1.4922,E1 25.1597,E2 448.1263} C_DIS
LIN {X 134.0025,Y 7.1013,Z 152,A -0.0951,B 24.9579,C -1.4999,E1 25.1595,E2 446.5453} C_DIS
Enddeposition()
END
